// TIA Portal V17 export
// export: Created 2025-03-07T09:18:18.4685776Z, ExportSetting WithDefaults, DisplayName Totally Integrated Automation Portal, DisplayVersion V17 Update 8, DisplayName TIA Portal Openness, DisplayVersion V17 Update 8, DisplayName TIA Portal Version Control Interface, DisplayVersion V17, DisplayName SINAMICS Startdrive Advanced, DisplayVersion V17 SP2, DisplayName SINAMICS Startdrive G110M, G120, G120C, G120D, G120P, G115D, DisplayVersion V17 SP2, DisplayName SINAMICS Startdrive G130, G150, S120, S150, SINAMICS MV, S210, DisplayVersion V17 SP2, DisplayName STEP 7 Professional, DisplayVersion V17 Update 8, DisplayName SINUMERIK ONE STEP 7 Toolbox, DisplayVersion V17 Update 12, DisplayName SINUMERIK 840D sl STEP 7 Toolbox, DisplayVersion V17 Update 12, DisplayName STEP 7 Safety, DisplayVersion V17 Update 6, DisplayName WinCC Advanced, DisplayVersion V17 Update 8
FUNCTION_BLOCK "FB1401_PNEUMATIC_SYSTEM"   // FB1401, LAD
{ S7_Optimized_Access := 'FALSE' }
AUTHOR : ETXETAR
VERSION : 1.0
// stored: AutoNumber false, IsIECCheckEnabled false, SetENOAutomatically false, UDAEnableTagReadback false
   VAR_INPUT
      OPTIONS_0 : Byte := 2#0000_0000;   // OPTIONS 0
      OPTIONS_1 : Byte := 2#0000_0000;   // OPTIONS 1
      OPTIONS_2 : Byte := 2#0000_0000;   // OPTIONS 1
      PRESSURE : Bool;   // PRESSURE INPUT
      DRIVE_UNBLOCKED : Bool;   // DRIVE UNBLOCKED INPUT
      CONNECTION_1_SENSOR : Bool;   // CONNECTION 1 SENSOR INPUT
      CONNECTION_2_SENSOR : Bool;   // CONNECTION 2 SENSOR INPUT
      FLOW_SENSOR : UInt;
      TEMPERATURE_SENSOR : UInt;
      PRESSURIZED : Bool;   // PRESSURIZED INPUT
      U01_GRIPPER_PRESSURIZED : Bool;   // UNIT 01 GRIPPER PRESSURIZED INPUT
      U01_LABERINT_PRESSURIZED : Bool;   // UNIT 01 LABERINT PRESSURIZED INPUT
      U01_UPPER_TABLE_PRESSURIZED : Bool;   // UNIT 01 UPPER TABLE PRESSURIZED INPUT
      U01_LOWER_TABLE_PRESSURIZED : Bool;   // UNIT 01 LOWER TABLE PRESSURIZED INPUT
      U01_CART_X_PRESSURIZED : Bool;   // UNIT 01 AXIS X CART PRESSURIZED INPUT
      U01_STA_3_MEAS_PRESSURIZED : Bool;   // UNIT 01 STATION 3 MEASURMENT UNIT PRESSURIZED INPUT
      U02_GRIPPER_PRESSURIZED : Bool;   // UNIT 02 GRIPPER PRESSURIZED INPUT
      U02_LABERINT_PRESSURIZED : Bool;   // UNIT 02 LABERINT PRESSURIZED INPUT
      U02_UPPER_TABLE_PRESSURIZED : Bool;   // UNIT 02 UPPER TABLE PRESSURIZED INPUT
      U02_LOWER_TABLE_PRESSURIZED : Bool;   // UNIT 02 LOWER TABLEPRESSURIZED INPUT
      U02_CART_X_PRESSURIZED : Bool;   // UNIT 02 AXIS X CART PRESSURIZED INPUT
      U02_STA_3_MEAS_PRESSURIZED : Bool;   // UNIT 02 STATION 3 MEASURMENT UNIT PRESSURIZED INPUT
      HMI_REQ_LINE : Bool;   // HMI REQUEST LINE
   END_VAR
   VAR_OUTPUT
      HMI_POWER_UP_COND_OFF : Bool;   // HMI POWER UP CONDITIONS OFF
      HMI_POWER_UP_COND_ON : Bool;   // HMI POWER UP CONDITIONS ON
      HMI_POWER_UP_EXECU_LEFT : Bool;   // HMI POWER UP EXECUTABLE LEFT
      HMI_POWER_UP_EXECU_RIGHT : Bool;   // HMI POWER UP EXECUTABLE RIGHT
      MAIN_VALVE : Bool;   // MAIN VALVE OUTPUT
      CONNECTION_1 : Bool;   // CONNECTION 1 OUTPUT
      CONNECTION_2 : Bool;   // CONNECTION 2 OUTPUT
      PRESSURIZATION_ON : Bool;   // PRESSURIZATION ON OUTPUT
      PRESSURIZATION_OFF : Bool;   // PRESSURIZATION OFF OUTPUT
      DRIVE_UNBLOCK : Bool;   // DRIVE UNBLOCK OUTPUT
   END_VAR
   VAR DB_SPECIFIC
      AIR_FLOW_VALUE : Real;   // AIR FLOW INPUT
      TEMPERATURE_VALUE : Real;   // TEMPERATURE INPUT VALUE
      PRESS_NOT_REACHED_ALARM : Bool;   // PRESSURE NOT REACHED ALARM
      PRESS_SWITCH_ALARM : Bool;   // PRESSURE SWITCH ALARM
      PRESS_MISSING_ALARM : Bool;   // PRESSURE MISSING ALARM
      CONNECTION_SENSOR_1_ALARM : Bool;   // CONNECTION SENSOR 1 ALARM
      CONNECTION_SENSOR_2_ALARM : Bool;   // CONNECTION SENSOR 2 ALARM
      UNBLOCK_DRIVE_PRESS_ALARM : Bool;   // UNBLOCK DRIVE PRESSURE ALARM
      UNBLOCK_DRIVE_PRESS_SWITCH_ALARM : Bool;   // UNBLOCK DRIVE PRESSURE SWITCH ALARM
      PRESSURIZATION_ALARM : Bool;   // PRESSURIZATION ALARM
      PRESSURIZATION_SWITCH_ALARM : Bool;   // PRESSURIZATION SWITCH ALARM
      PNEUMATIC_TEMPERATURE_INPUT_ALARM : Bool;   // PNEUMATIC INPUT TEMPERATURE ALARM
      PNEUMATIC_FLOW_INPUT_ALARM : Bool;   // PNEUMATIC INPUT FLOW ALARM
      U01_GRIPPER_PRESSURIZATION_ALARM : Bool;   // UNIT 01 GRIPPER PRESSURIZATION ALARM
      U01_GRIPPER_PRESSURIZATION_SWITCH_ALARM : Bool;   // UNIT 01 GRIPPER PRESSURIZATION SWITCH ALARM
      U01_LABERINT_PRESSURIZATION_ALARM : Bool;   // UNIT 01 LABERINT PRESSURIZATION ALARM
      U01_LABERINT_PRESSURIZATION_SWITCH_ALARM : Bool;   // UNIT 01 LABERINT PRESSURIZATION SWITCH ALARM
      U01_UPPER_TABLE_PRESSURIZATION_ALARM : Bool;   // UNIT 01 UPPER TABLE PRESSURIZATION ALARM
      U01_UPPER_TABLE_PRESSURIZATION_SWITCH_ALARM : Bool;   // UNIT 01 UPPER TABLE PRESSURIZATION SWITCH ALARM
      U01_LOWER_TABLE_PRESSURIZATION_ALARM : Bool;   // UNIT 01 LOWER TABLE PRESSURIZATION ALARM
      U01_LOWER_TABLE_PRESSURIZATION_SWITCH_ALARM : Bool;   // UNIT 01 LOWER TABLE PRESSURIZATION SWITCH ALARM
      U01_CART_AXIS_X_PRESSURIZATION_ALARM : Bool;   // UNIT 01 CART AXIS X PRESSURIZATION ALARM
      U01_CART_AXIS_X_PRESSURIZATION_SWITCH_ALARM : Bool;   // UNIT 01 CART AXIS X PRESSURIZATION SWITCH ALARM
      U01_STA_3_MEAS_PRESSURIZATION_ALARM : Bool;   // UNIT 01 STATION 3 MEASUREMENT UNIT PRESSURIZATION ALARM
      U01_STA_3_MEAS_PRESSURIZATION_SWITCH_ALARM : Bool;   // UNIT 01 STATION 3 MEASUREMENT UNIT PRESSURIZATION SWITCH ALARM
      U02_GRIPPER_PRESSURIZATION_ALARM : Bool;   // UNIT 02 GRIPPER PRESSURIZATION ALARM
      U02_GRIPPER_PRESSURIZATION_SWITCH_ALARM : Bool;   // UNIT 02 GRIPPER PRESSURIZATION SWITCH ALARM
      U02_LABERINT_PRESSURIZATION_ALARM : Bool;   // UNIT 02 LABERINT PRESSURIZATION ALARM
      U02_LABERINT_PRESSURIZATION_SWITCH_ALARM : Bool;   // UNIT 02 LABERINT PRESSURIZATION SWITCH ALARM
      U02_UPPER_TABLE_PRESSURIZATION_ALARM : Bool;   // UNIT 02 UPPER TABLE PRESSURIZATION ALARM
      U02_UPPER_TABLE_PRESSURIZATION_SWITCH_ALARM : Bool;   // UNIT 02 UPPER TABLE PRESSURIZATION SWITCH ALARM
      U02_LOWER_TABLE_PRESSURIZATION_ALARM : Bool;   // UNIT 02 LOWER TABLE PRESSURIZATION ALARM
      U02_LOWER_TABLE_PRESSURIZATION_SWITCH_ALARM : Bool;   // UNIT 02 LOWER TABLE PRESSURIZATION SWITCH ALARM
      U02_CART_AXIS_X_PRESSURIZATION_ALARM : Bool;   // UNIT 02 CART AXIS X PRESSURIZATION ALARM
      U02_CART_AXIS_X_PRESSURIZATION_SWITCH_ALARM : Bool;   // UNIT 02 CART AXIS X PRESSURIZATION SWITCH ALARM
      U02_STA_3_MEAS_PRESSURIZATION_ALARM : Bool;   // UNIT 02 STATION 3 MEASUREMENT UNIT PRESSURIZATION ALARM
      U02_STA_3_MEAS_PRESSURIZATION_SWITCH_ALARM : Bool;   // UNIT 02 STATION 3 MEASUREMENT UNIT PRESSURIZATION SWITCH ALARM
      SWITCH_ON_GENERAL_CONDITIONS : Bool;   // SWITCH ON GENERAL CONDITIONS
      SWITCH_ON_INITIAL_CONDITIONS : Bool;   // SWITCH ON INITIAL CONDITIONS
      SWITCH_ON_MANUAL_REQUEST : Bool;   // SWITCH ON MANUAL REQUEST
      SWITCH_ON_AUTO_REQUEST : Bool;   // SWITCH ON AUTO REQUEST
      SWITCH_ON_GLOBAL_REQUEST : Bool;   // SWITCH ON GLOBAL REQUEST
      SWITCH_ON_COMMAND : Bool;   // SWITCH ON COMMAND
      SWITCH_ON : Bool;   // SWITCH ON
      IN_SERVICE : Bool;   // IN SERVICE
      SWITCH_OFF_GENERAL_CONDITIONS : Bool;   // SWITCH OFF GENERAL CONDITIONS
      SWITCH_OFF_INITIAL_CONDITIONS : Bool;   // SWITCH OFF INITIAL CONDITIONS
      SWITCH_OFF_MANUAL_REQUEST : Bool;   // SWITCH OFF MANUAL REQUEST
      SWITCH_OFF_AUTO_REQUEST : Bool;   // SWITCH OFF AUTO REQUEST
      SWITCH_OFF_GLOBAL_REQUEST : Bool;   // SWITCH OFF GLOBAL REQUEST
      SWITCH_OFF_COMMAND : Bool;   // SWITCH OFF COMMAND
      SWITCH_OFF : Bool;   // SWITCH OFF
      OUT_OF_SERVICE : Bool;   // OUT OF SERVICE
      MANUAL_REQUEST_HELP : Bool;   // MANUAL REQUEST HELP
      SWITCH_ON_GENERAL_CONDITION_HELP : Bool;   // SWITCH ON GENERAL CONDITION HELP
      SWITCH_ON_INITIAL_CONDITION_HELP : Bool;   // SWITCH ON INITIAL CONDITION HELP
      SWITCH_OFF_GENERAL_CONDITION_HELP : Bool;   // SWITCH OFF GENERAL CONDITION HELP
      SWITCH_OFF_INITIAL_CONDITION_HELP : Bool;   // SWITCH OFF INITIAL CONDITION HELP
      ANY_ACTIVE_ALARM : Bool;   // ANY ACTIVE ALARM
      IS_ALARMS : Bool;   // IMMEDIATE STOP ALARMS
      SEOC_ALARMS : Bool;   // STOP END OF CYCLE ALARMS
      WARNINGS : Bool;   // WARNINGS
      WARNINGS_GONE : Bool;   // WARNINGS GONE
      TIMER_PRESSURE_ALARM : TON_TIME;   // PRESSURE TIMER
      TIMER_PRESSURE_SWITCH_ALARM : TON_TIME;   // PRESSURE SWITCH TIMER
      TIMER_PRESSURE_MISSING_ALARM : TON_TIME;   // PRESSURE MISSING TIMER
      TIMER_CONNECTION_SENSOR_1_ALARM : TON_TIME;   // CONNECTION SENSOR 1 TIMER
      TIMER_CONNECTION_SENSOR_1_SWITCH_ALARM : TON_TIME;   // CONNECTION SENSOR 1 SWITCH TIMER
      TIMER_CONNECTION_SENSOR_2_ALARM : TON_TIME;   // CONNECTION SENSOR 2 TIMER
      TIMER_CONNECTION_SENSOR_2_SWITCH_ALARM : TON_TIME;   // CONNECTION SENSOR 2 SWITCH TIMER
      TIMER_DRIVE_PRESSURE_UNBLOCK_ALARM : TON_TIME;   // DRIVE PRESSURE UNBLOCK TIMER
      TIMER_DRIVE_PRESSURE_UNBLOCK_SWITCH_ALARM : TON_TIME;   // DRIVE PRESSURE UNBLOCK SWITCH TIMER
      TIMER_PRESSURE_ON_DEVICES : TON_TIME;   // PRESSURE ON DEVICES TIMER
      TIMER_PRESSURE_OFF_DEVICES : TON_TIME;   // PRESSURE OFF DEVICES TIMER
      TIMER_PRESSURIZATION_OFF_DELAY { S7_SetPoint := 'True'} : TOF_TIME;
   END_VAR
   VAR_TEMP
      INPUTS_MASK : Byte;   // INPUT MASK
      O_BYTE_0 : Struct   // OPTIONS BYTE 0
         PRESSURE_PRESENT : Bool;   // PRESSURE PRESENT OPTION
         CONNECTION_SENSOR_1 : Bool;   // CONNECTION SENSOR 1 OPTION
         CONNECTION_SENSOR_2 : Bool;   // CONNECTION SENSOR 2 OPTION
         UNBLOCK_DRIVE_VALVE : Bool;   // DRIVE VALVE OPTION
         PRESSURIZED : Bool;   // PRESSURIZED OPTION
         U01_GRIPPER_PRESSURIZED : Bool;   // UNIT 01 GRIPPER PRESSURIZED OPTION
         U01_LABERINT_PRESSURIZED : Bool;   // UNIT 01 LABERINT PRESSURIZED OPTION
         U01_UPPER_TABLE_PRESSURIZED : Bool;   // UNIT 01 UPPER TABLE PRESSURIZED OPTION
      END_STRUCT;
      O_BYTE_1 : Struct   // OPTIONS BYTE 1
         U01_LOWER_TABLE_PRESSURIZED : Bool;   // UNIT 01 LOWER TABLE PRESSURIZED OPTION
         U01_X_CART_PRESSURIZED : Bool;   // UNIT 01 AXIS X CART PRESSURIZED OPTION
         U01_STA_3_MEAS_PRESSURIZED : Bool;   // UNIT 01 STATION 3 MEASUREMENT PRESSURIZED OPTION
         U01_STA_4_MEAS_PRESSURIZED : Bool;   // UNIT 01 STATION 4 MEASUREMENT PRESSURIZED OPTION
         U02_GRIPPER_PRESSURIZED : Bool;   // UNIT 02 GRIPPER PRESSURIZED OPTION
         U02_LABERINT_PRESSURIZED : Bool;   // UNIT 02 LABERINT PRESSURIZED OPTION
         U02_UPPER_TABLE_PRESSURIZED : Bool;   // UNIT 02 UPPER TABLE PRESSURIZED OPTION
         U02_LOWER_TABLE_PRESSURIZED : Bool;   // UNIT 02 LOWER TABLE PRESSURIZED OPTION
      END_STRUCT;
      O_BYTE_2 : Struct   // OPTIONS BYTE 1
         U02_X_CART_PRESSURIZED : Bool;   // UNIT 02 AXIS X CART PRESSURIZED OPTION
         U02_STA_3_MEAS_PRESSURIZED : Bool;   // UNIT 02 STATION 3 MEASUREMENT PRESSURIZED OPTION
         U02_STA_4_MEAS_PRESSURIZED : Bool;   // UNIT 02 STATION 4 MEASUREMENT PRESSURIZED OPTION
         INPUT_FLOW_OPTION : Bool;   // INPUT FLOW OPTION
         INPUT_TEMPERATURE_OPTION : Bool;   // INPUT TEMPERATURE OPTION
         SPARE_5 : Bool;   // SPARE OPTION
         SPARE_6 : Bool;   // SPARE OPTION
         SPARE_7 : Bool;   // SPARE OPTION
      END_STRUCT;
      TEMPERATURE_TEMP : UInt;   // TEMPERATURE TEMPORAL
      PRESSURE_ON_DELAYED : Bool;   // PRESSURE ON DELAYED
      PRESSURE_OFF_DELAYED : Bool;   // PRESSURE OFF DELAYED
      DB_NUMBER : DInt;   // DB NUMBER FOR ALARM DECODING
   END_VAR
   // TIMER_PRESSURE_ALARM.PT := T#1M;
   // TIMER_PRESSURE_SWITCH_ALARM.PT := T#1M;
   // TIMER_PRESSURE_MISSING_ALARM.PT := T#1s;
   // TIMER_CONNECTION_SENSOR_1_ALARM.PT := T#1s;
   // TIMER_CONNECTION_SENSOR_1_SWITCH_ALARM.PT := T#1s;
   // TIMER_CONNECTION_SENSOR_2_ALARM.PT := T#1s;
   // TIMER_CONNECTION_SENSOR_2_SWITCH_ALARM.PT := T#1s;
   // TIMER_DRIVE_PRESSURE_UNBLOCK_ALARM.PT := T#3s;
   // TIMER_DRIVE_PRESSURE_UNBLOCK_SWITCH_ALARM.PT := T#3s;
   // TIMER_PRESSURE_ON_DEVICES.PT := T#5s;
   // TIMER_PRESSURE_OFF_DEVICES.PT := T#31M;
   // TIMER_PRESSURIZATION_OFF_DELAY.PT := T#30M;
   VAR_TEMP   // added for the SCL form of the ladder/FBD networks
      _w1 : Bool;
   END_VAR
BEGIN

NETWORK
TITLE = READ INSTANCE DB
      L     DINO;
      +     10#800000;
      T     #DB_NUMBER;


REGION Network 2: OPTIONS
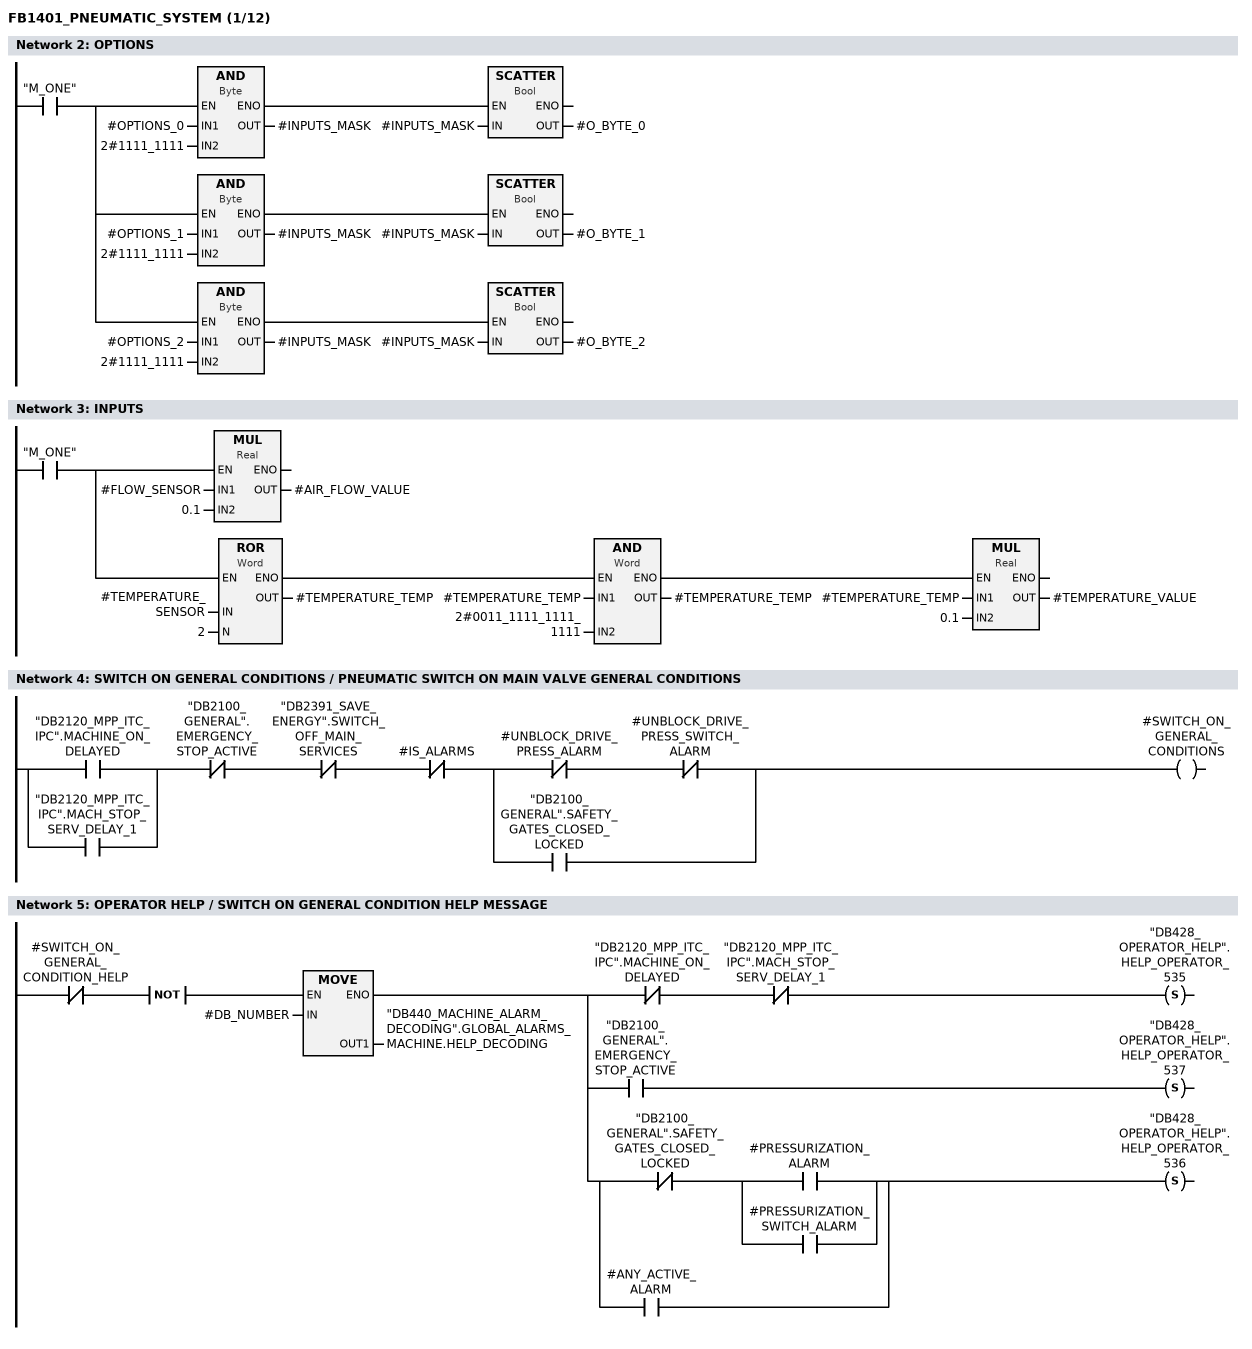
   RUNG wire#powerrail
      Contact( "M_ONE" )
      wire#w1
      { S7_Templates := "SrcType := Byte"; S7_GenerateENO := "TRUE" } And(in1 := #OPTIONS_0, in2 := 2#1111_1111, out => #INPUTS_MASK)
      { S7_Templates := "[dest_type := Bool, src_type := Byte]" } SCATTER(IN := #INPUTS_MASK, OUT => #O_BYTE_0)
   END_RUNG
   RUNG wire#w1
      { S7_Templates := "SrcType := Byte"; S7_GenerateENO := "TRUE" } And(in1 := #OPTIONS_1, in2 := 2#1111_1111, out => #INPUTS_MASK)
      { S7_Templates := "[dest_type := Bool, src_type := Byte]" } SCATTER(IN := #INPUTS_MASK, OUT => #O_BYTE_1)
   END_RUNG
   RUNG wire#w1
      { S7_Templates := "SrcType := Byte"; S7_GenerateENO := "TRUE" } And(in1 := #OPTIONS_2, in2 := 2#1111_1111, out => #INPUTS_MASK)
      { S7_Templates := "[dest_type := Bool, src_type := Byte]" } SCATTER(IN := #INPUTS_MASK, OUT => #O_BYTE_2)
   END_RUNG
   // the same network as SCL:
   IF "M_ONE" THEN #INPUTS_MASK := #OPTIONS_0 AND 2#1111_1111; END_IF;
   #_w1 := "M_ONE";
   IF #_w1 THEN
       SCATTER(IN := #INPUTS_MASK, OUT => #O_BYTE_0);
       #INPUTS_MASK := #OPTIONS_1 AND 2#1111_1111;
       SCATTER(IN := #INPUTS_MASK, OUT => #O_BYTE_1);
       #INPUTS_MASK := #OPTIONS_2 AND 2#1111_1111;
       SCATTER(IN := #INPUTS_MASK, OUT => #O_BYTE_2);
   END_IF;
END_REGION

REGION Network 3: INPUTS
   IF "M_ONE" THEN
       #AIR_FLOW_VALUE := #FLOW_SENSOR * 0.1;
       #TEMPERATURE_TEMP := ROR(IN := #TEMPERATURE_SENSOR, N := 2);
       #TEMPERATURE_TEMP := #TEMPERATURE_TEMP AND 2#0011_1111_1111_1111;
       #TEMPERATURE_VALUE := #TEMPERATURE_TEMP * 0.1;
   END_IF;
END_REGION

REGION Network 4: SWITCH ON GENERAL CONDITIONS / PNEUMATIC SWITCH ON MAIN VALVE GENERAL CONDITIONS
   RUNG wire#powerrail
      Contact( "DB2120_MPP_ITC_IPC".MACHINE_ON_DELAYED )
      wire#w1
      I_Contact( "DB2100_GENERAL".EMERGENCY_STOP_ACTIVE )
      I_Contact( "DB2391_SAVE_ENERGY".SWITCH_OFF_MAIN_SERVICES )
      I_Contact( #IS_ALARMS )
      wire#w2
      I_Contact( #UNBLOCK_DRIVE_PRESS_ALARM )
      I_Contact( #UNBLOCK_DRIVE_PRESS_SWITCH_ALARM )
      wire#w3
      Coil( #SWITCH_ON_GENERAL_CONDITIONS )
   END_RUNG
   RUNG wire#powerrail
      Contact( "DB2120_MPP_ITC_IPC".MACH_STOP_SERV_DELAY_1 )
   END_RUNG wire#w1
   RUNG wire#w2
      Contact( "DB2100_GENERAL".SAFETY_GATES_CLOSED_LOCKED )
   END_RUNG wire#w3
   // the same network as SCL:
   #SWITCH_ON_GENERAL_CONDITIONS := ("DB2120_MPP_ITC_IPC".MACHINE_ON_DELAYED OR "DB2120_MPP_ITC_IPC".MACH_STOP_SERV_DELAY_1) AND NOT "DB2100_GENERAL".EMERGENCY_STOP_ACTIVE AND NOT "DB2391_SAVE_ENERGY".SWITCH_OFF_MAIN_SERVICES AND NOT #IS_ALARMS AND ((NOT #UNBLOCK_DRIVE_PRESS_ALARM AND NOT #UNBLOCK_DRIVE_PRESS_SWITCH_ALARM) OR "DB2100_GENERAL".SAFETY_GATES_CLOSED_LOCKED);
END_REGION

REGION Network 5: OPERATOR HELP / SWITCH ON GENERAL CONDITION HELP MESSAGE
   RUNG wire#powerrail
      I_Contact( #SWITCH_ON_GENERAL_CONDITION_HELP )
      Not()
      { S7_GenerateENO := "TRUE" } Move(in := #DB_NUMBER, out1 => "DB440_MACHINE_ALARM_DECODING".GLOBAL_ALARMS_MACHINE.HELP_DECODING)
      wire#w1
      I_Contact( "DB2120_MPP_ITC_IPC".MACHINE_ON_DELAYED )
      I_Contact( "DB2120_MPP_ITC_IPC".MACH_STOP_SERV_DELAY_1 )
      S_Coil( "DB428_OPERATOR_HELP".HELP_OPERATOR_535 )
   END_RUNG
   RUNG wire#w1
      Contact( "DB2100_GENERAL".EMERGENCY_STOP_ACTIVE )
      S_Coil( "DB428_OPERATOR_HELP".HELP_OPERATOR_537 )
   END_RUNG
   RUNG wire#w1
      I_Contact( "DB2100_GENERAL".SAFETY_GATES_CLOSED_LOCKED )
      wire#w2
      Contact( #PRESSURIZATION_ALARM )
      wire#w3
      S_Coil( "DB428_OPERATOR_HELP".HELP_OPERATOR_536 )
   END_RUNG
   RUNG wire#w2
      Contact( #PRESSURIZATION_SWITCH_ALARM )
   END_RUNG wire#w3
   RUNG wire#w1
      Contact( #ANY_ACTIVE_ALARM )
   END_RUNG wire#w3
   // the same network as SCL:
   // ENO of a box is taken as its EN; it also drops when the box reports an error
   #_w1 := NOT (NOT #SWITCH_ON_GENERAL_CONDITION_HELP);
   IF #_w1 THEN "DB440_MACHINE_ALARM_DECODING".GLOBAL_ALARMS_MACHINE.HELP_DECODING := #DB_NUMBER; END_IF;
   IF #_w1 AND NOT "DB2120_MPP_ITC_IPC".MACHINE_ON_DELAYED AND NOT "DB2120_MPP_ITC_IPC".MACH_STOP_SERV_DELAY_1 THEN
       "DB428_OPERATOR_HELP".HELP_OPERATOR_535 := TRUE;
   END_IF;
   IF #_w1 AND "DB2100_GENERAL".EMERGENCY_STOP_ACTIVE THEN
       "DB428_OPERATOR_HELP".HELP_OPERATOR_537 := TRUE;
   END_IF;
   IF #_w1 AND ((NOT "DB2100_GENERAL".SAFETY_GATES_CLOSED_LOCKED AND (#PRESSURIZATION_ALARM OR #PRESSURIZATION_SWITCH_ALARM)) OR #ANY_ACTIVE_ALARM) THEN
       "DB428_OPERATOR_HELP".HELP_OPERATOR_536 := TRUE;
   END_IF;
END_REGION

REGION Network 6: SWITCH ON INITIAL CONDITIONS
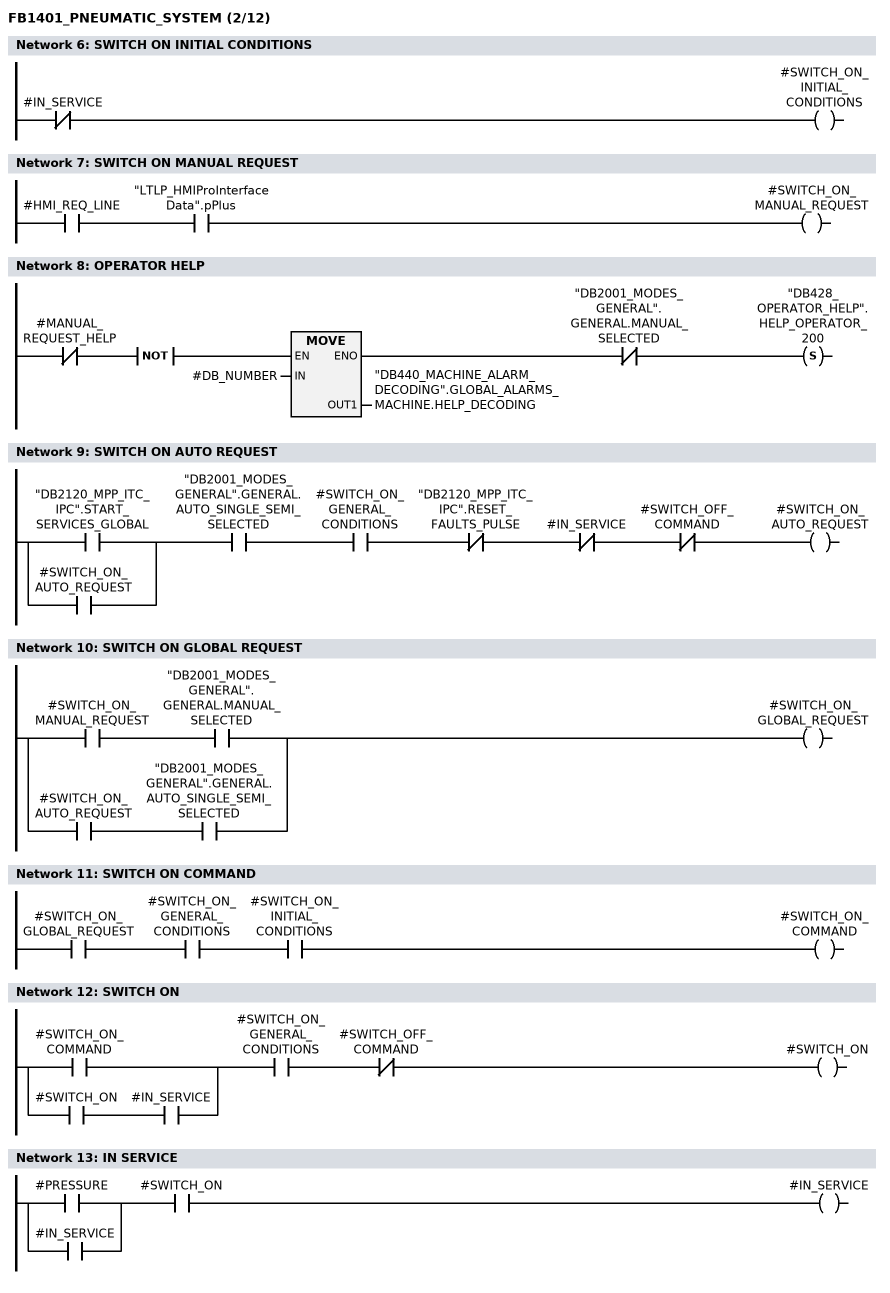
   RUNG wire#powerrail
      I_Contact( #IN_SERVICE )
      Coil( #SWITCH_ON_INITIAL_CONDITIONS )
   END_RUNG
   // the same network as SCL:
   #SWITCH_ON_INITIAL_CONDITIONS := NOT #IN_SERVICE;
END_REGION

REGION Network 7: SWITCH ON MANUAL REQUEST
   RUNG wire#powerrail
      Contact( #HMI_REQ_LINE )
      Contact( "LTLP_HMIProInterfaceData".pPlus )
      Coil( #SWITCH_ON_MANUAL_REQUEST )
   END_RUNG
   // the same network as SCL:
   #SWITCH_ON_MANUAL_REQUEST := #HMI_REQ_LINE AND "LTLP_HMIProInterfaceData".pPlus;
END_REGION

REGION Network 8: OPERATOR HELP
   RUNG wire#powerrail
      I_Contact( #MANUAL_REQUEST_HELP )
      Not()
      { S7_GenerateENO := "TRUE" } Move(in := #DB_NUMBER, out1 => "DB440_MACHINE_ALARM_DECODING".GLOBAL_ALARMS_MACHINE.HELP_DECODING)
      I_Contact( "DB2001_MODES_GENERAL".GENERAL.MANUAL_SELECTED )
      S_Coil( "DB428_OPERATOR_HELP".HELP_OPERATOR_200 )
   END_RUNG
   // the same network as SCL:
   // ENO of a box is taken as its EN; it also drops when the box reports an error
   #_w1 := NOT (NOT #MANUAL_REQUEST_HELP);
   IF #_w1 THEN "DB440_MACHINE_ALARM_DECODING".GLOBAL_ALARMS_MACHINE.HELP_DECODING := #DB_NUMBER; END_IF;
   IF #_w1 AND NOT "DB2001_MODES_GENERAL".GENERAL.MANUAL_SELECTED THEN
       "DB428_OPERATOR_HELP".HELP_OPERATOR_200 := TRUE;
   END_IF;
END_REGION

REGION Network 9: SWITCH ON AUTO REQUEST
   RUNG wire#powerrail
      Contact( "DB2120_MPP_ITC_IPC".START_SERVICES_GLOBAL )
      wire#w1
      Contact( "DB2001_MODES_GENERAL".GENERAL.AUTO_SINGLE_SEMI_SELECTED )
      Contact( #SWITCH_ON_GENERAL_CONDITIONS )
      I_Contact( "DB2120_MPP_ITC_IPC".RESET_FAULTS_PULSE )
      I_Contact( #IN_SERVICE )
      I_Contact( #SWITCH_OFF_COMMAND )
      Coil( #SWITCH_ON_AUTO_REQUEST )
   END_RUNG
   RUNG wire#powerrail
      Contact( #SWITCH_ON_AUTO_REQUEST )
   END_RUNG wire#w1
   // the same network as SCL:
   #SWITCH_ON_AUTO_REQUEST := ("DB2120_MPP_ITC_IPC".START_SERVICES_GLOBAL OR #SWITCH_ON_AUTO_REQUEST) AND "DB2001_MODES_GENERAL".GENERAL.AUTO_SINGLE_SEMI_SELECTED AND #SWITCH_ON_GENERAL_CONDITIONS AND NOT "DB2120_MPP_ITC_IPC".RESET_FAULTS_PULSE AND NOT #IN_SERVICE AND NOT #SWITCH_OFF_COMMAND;
END_REGION

REGION Network 10: SWITCH ON GLOBAL REQUEST
   RUNG wire#powerrail
      Contact( #SWITCH_ON_MANUAL_REQUEST )
      Contact( "DB2001_MODES_GENERAL".GENERAL.MANUAL_SELECTED )
      wire#w1
      Coil( #SWITCH_ON_GLOBAL_REQUEST )
   END_RUNG
   RUNG wire#powerrail
      Contact( #SWITCH_ON_AUTO_REQUEST )
      Contact( "DB2001_MODES_GENERAL".GENERAL.AUTO_SINGLE_SEMI_SELECTED )
   END_RUNG wire#w1
   // the same network as SCL:
   #SWITCH_ON_GLOBAL_REQUEST := (#SWITCH_ON_MANUAL_REQUEST AND "DB2001_MODES_GENERAL".GENERAL.MANUAL_SELECTED) OR (#SWITCH_ON_AUTO_REQUEST AND "DB2001_MODES_GENERAL".GENERAL.AUTO_SINGLE_SEMI_SELECTED);
END_REGION

REGION Network 11: SWITCH ON COMMAND
   RUNG wire#powerrail
      Contact( #SWITCH_ON_GLOBAL_REQUEST )
      Contact( #SWITCH_ON_GENERAL_CONDITIONS )
      Contact( #SWITCH_ON_INITIAL_CONDITIONS )
      Coil( #SWITCH_ON_COMMAND )
   END_RUNG
   // the same network as SCL:
   #SWITCH_ON_COMMAND := #SWITCH_ON_GLOBAL_REQUEST AND #SWITCH_ON_GENERAL_CONDITIONS AND #SWITCH_ON_INITIAL_CONDITIONS;
END_REGION

REGION Network 12: SWITCH ON
   RUNG wire#powerrail
      Contact( #SWITCH_ON_COMMAND )
      wire#w1
      Contact( #SWITCH_ON_GENERAL_CONDITIONS )
      I_Contact( #SWITCH_OFF_COMMAND )
      Coil( #SWITCH_ON )
   END_RUNG
   RUNG wire#powerrail
      Contact( #SWITCH_ON )
      Contact( #IN_SERVICE )
   END_RUNG wire#w1
   // the same network as SCL:
   #SWITCH_ON := (#SWITCH_ON_COMMAND OR (#SWITCH_ON AND #IN_SERVICE)) AND #SWITCH_ON_GENERAL_CONDITIONS AND NOT #SWITCH_OFF_COMMAND;
END_REGION

REGION Network 13: IN SERVICE
   RUNG wire#powerrail
      Contact( #PRESSURE )
      wire#w1
      Contact( #SWITCH_ON )
      Coil( #IN_SERVICE )
   END_RUNG
   RUNG wire#powerrail
      Contact( #IN_SERVICE )
   END_RUNG wire#w1
   // the same network as SCL:
   #IN_SERVICE := (#PRESSURE OR #IN_SERVICE) AND #SWITCH_ON;
END_REGION

REGION Network 14: SWITCH OFF GENERAL CONDITIONS
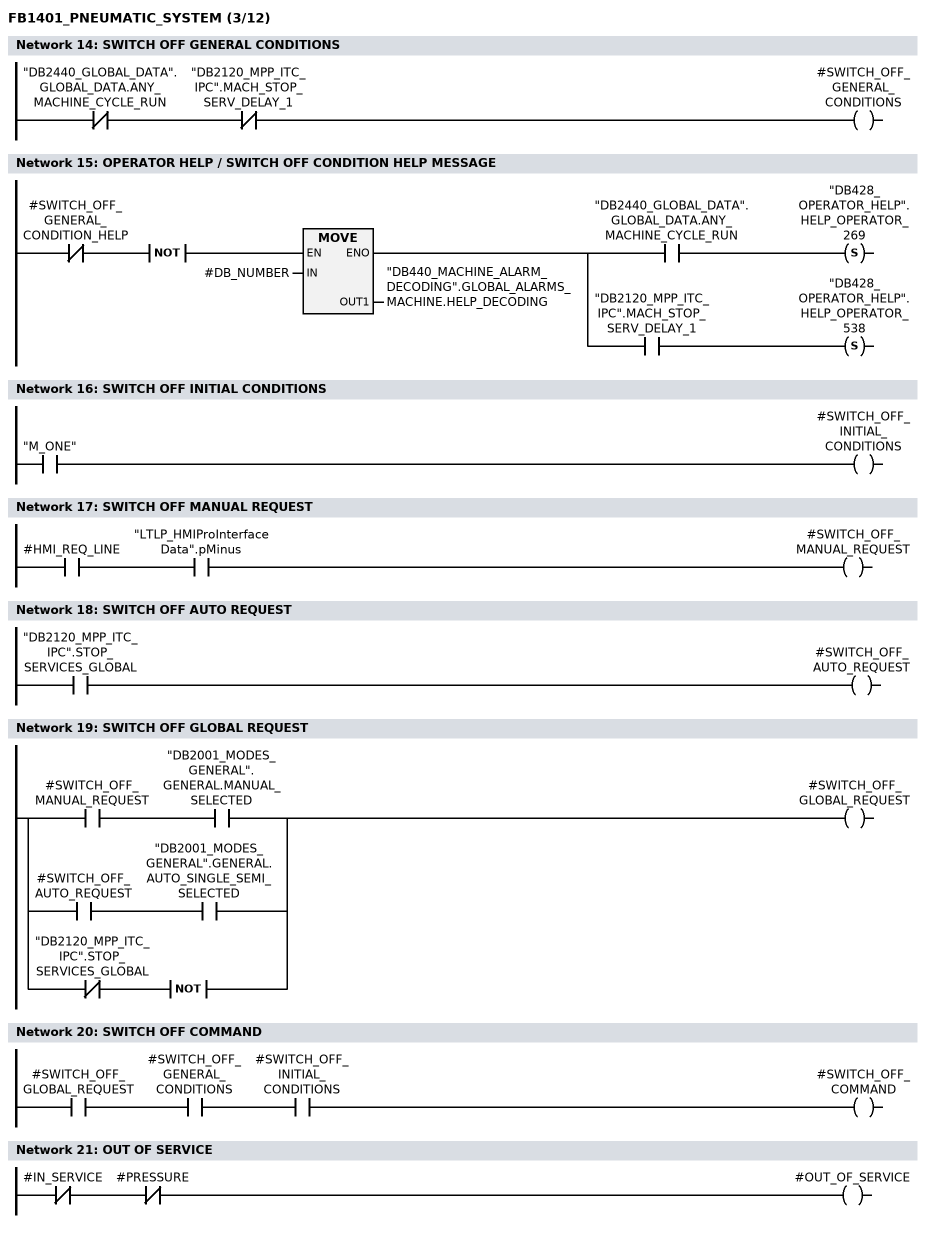
   RUNG wire#powerrail
      I_Contact( "DB2440_GLOBAL_DATA".GLOBAL_DATA.ANY_MACHINE_CYCLE_RUN )
      I_Contact( "DB2120_MPP_ITC_IPC".MACH_STOP_SERV_DELAY_1 )
      Coil( #SWITCH_OFF_GENERAL_CONDITIONS )
   END_RUNG
   // the same network as SCL:
   #SWITCH_OFF_GENERAL_CONDITIONS := NOT "DB2440_GLOBAL_DATA".GLOBAL_DATA.ANY_MACHINE_CYCLE_RUN AND NOT "DB2120_MPP_ITC_IPC".MACH_STOP_SERV_DELAY_1;
END_REGION

REGION Network 15: OPERATOR HELP / SWITCH OFF CONDITION HELP MESSAGE
   RUNG wire#powerrail
      I_Contact( #SWITCH_OFF_GENERAL_CONDITION_HELP )
      Not()
      { S7_GenerateENO := "TRUE" } Move(in := #DB_NUMBER, out1 => "DB440_MACHINE_ALARM_DECODING".GLOBAL_ALARMS_MACHINE.HELP_DECODING)
      wire#w1
      Contact( "DB2440_GLOBAL_DATA".GLOBAL_DATA.ANY_MACHINE_CYCLE_RUN )
      S_Coil( "DB428_OPERATOR_HELP".HELP_OPERATOR_269 )
   END_RUNG
   RUNG wire#w1
      Contact( "DB2120_MPP_ITC_IPC".MACH_STOP_SERV_DELAY_1 )
      S_Coil( "DB428_OPERATOR_HELP".HELP_OPERATOR_538 )
   END_RUNG
   // the same network as SCL:
   // ENO of a box is taken as its EN; it also drops when the box reports an error
   #_w1 := NOT (NOT #SWITCH_OFF_GENERAL_CONDITION_HELP);
   IF #_w1 THEN "DB440_MACHINE_ALARM_DECODING".GLOBAL_ALARMS_MACHINE.HELP_DECODING := #DB_NUMBER; END_IF;
   IF #_w1 AND "DB2440_GLOBAL_DATA".GLOBAL_DATA.ANY_MACHINE_CYCLE_RUN THEN
       "DB428_OPERATOR_HELP".HELP_OPERATOR_269 := TRUE;
   END_IF;
   IF #_w1 AND "DB2120_MPP_ITC_IPC".MACH_STOP_SERV_DELAY_1 THEN
       "DB428_OPERATOR_HELP".HELP_OPERATOR_538 := TRUE;
   END_IF;
END_REGION

REGION Network 16: SWITCH OFF INITIAL CONDITIONS
   RUNG wire#powerrail
      Contact( "M_ONE" )
      Coil( #SWITCH_OFF_INITIAL_CONDITIONS )
   END_RUNG
   // the same network as SCL:
   #SWITCH_OFF_INITIAL_CONDITIONS := "M_ONE";
END_REGION

REGION Network 17: SWITCH OFF MANUAL REQUEST
   RUNG wire#powerrail
      Contact( #HMI_REQ_LINE )
      Contact( "LTLP_HMIProInterfaceData".pMinus )
      Coil( #SWITCH_OFF_MANUAL_REQUEST )
   END_RUNG
   // the same network as SCL:
   #SWITCH_OFF_MANUAL_REQUEST := #HMI_REQ_LINE AND "LTLP_HMIProInterfaceData".pMinus;
END_REGION

REGION Network 18: SWITCH OFF AUTO REQUEST
   RUNG wire#powerrail
      Contact( "DB2120_MPP_ITC_IPC".STOP_SERVICES_GLOBAL )
      Coil( #SWITCH_OFF_AUTO_REQUEST )
   END_RUNG
   // the same network as SCL:
   #SWITCH_OFF_AUTO_REQUEST := "DB2120_MPP_ITC_IPC".STOP_SERVICES_GLOBAL;
END_REGION

REGION Network 19: SWITCH OFF GLOBAL REQUEST
   RUNG wire#powerrail
      Contact( #SWITCH_OFF_MANUAL_REQUEST )
      Contact( "DB2001_MODES_GENERAL".GENERAL.MANUAL_SELECTED )
      wire#w1
      Coil( #SWITCH_OFF_GLOBAL_REQUEST )
   END_RUNG
   RUNG wire#powerrail
      Contact( #SWITCH_OFF_AUTO_REQUEST )
      Contact( "DB2001_MODES_GENERAL".GENERAL.AUTO_SINGLE_SEMI_SELECTED )
   END_RUNG wire#w1
   RUNG wire#powerrail
      I_Contact( "DB2120_MPP_ITC_IPC".STOP_SERVICES_GLOBAL )
      Not()
   END_RUNG wire#w1
   // the same network as SCL:
   #SWITCH_OFF_GLOBAL_REQUEST := (#SWITCH_OFF_MANUAL_REQUEST AND "DB2001_MODES_GENERAL".GENERAL.MANUAL_SELECTED) OR (#SWITCH_OFF_AUTO_REQUEST AND "DB2001_MODES_GENERAL".GENERAL.AUTO_SINGLE_SEMI_SELECTED) OR NOT (NOT "DB2120_MPP_ITC_IPC".STOP_SERVICES_GLOBAL);
END_REGION

REGION Network 20: SWITCH OFF COMMAND
   RUNG wire#powerrail
      Contact( #SWITCH_OFF_GLOBAL_REQUEST )
      Contact( #SWITCH_OFF_GENERAL_CONDITIONS )
      Contact( #SWITCH_OFF_INITIAL_CONDITIONS )
      Coil( #SWITCH_OFF_COMMAND )
   END_RUNG
   // the same network as SCL:
   #SWITCH_OFF_COMMAND := #SWITCH_OFF_GLOBAL_REQUEST AND #SWITCH_OFF_GENERAL_CONDITIONS AND #SWITCH_OFF_INITIAL_CONDITIONS;
END_REGION

REGION Network 21: OUT OF SERVICE
   RUNG wire#powerrail
      I_Contact( #IN_SERVICE )
      I_Contact( #PRESSURE )
      Coil( #OUT_OF_SERVICE )
   END_RUNG
   // the same network as SCL:
   #OUT_OF_SERVICE := NOT #IN_SERVICE AND NOT #PRESSURE;
END_REGION

REGION Network 22: PRESSURE NOT REACHED ALARM / PNEUMATIC SYSTEM PRESSURE SWITCH ALARM
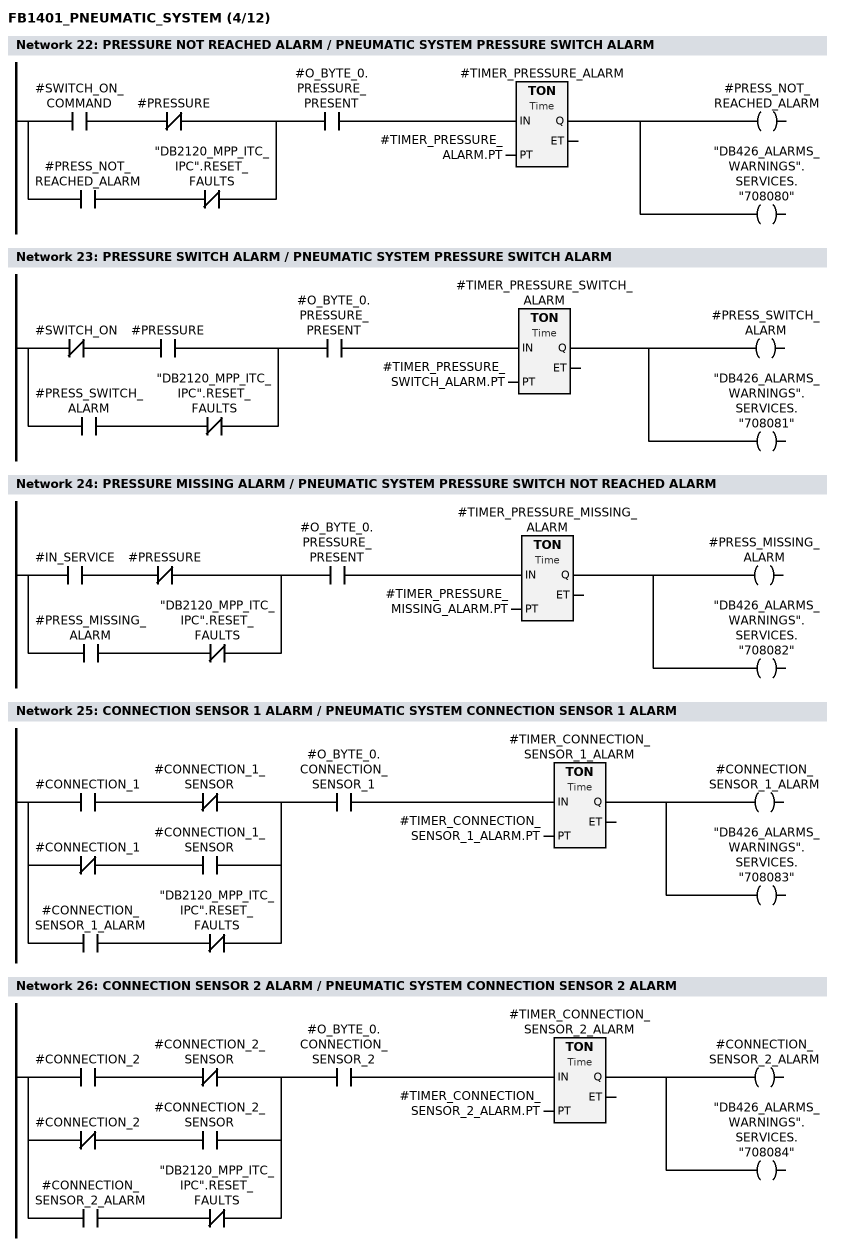
   RUNG wire#powerrail
      Contact( #SWITCH_ON_COMMAND )
      I_Contact( #PRESSURE )
      wire#w1
      Contact( #O_BYTE_0.PRESSURE_PRESENT )
      { S7_Templates := "time_type := Time" } #TIMER_PRESSURE_ALARM.TON(pt := #TIMER_PRESSURE_ALARM.PT, et =>)
      wire#w2
      Coil( #PRESS_NOT_REACHED_ALARM )
   END_RUNG
   RUNG wire#powerrail
      Contact( #PRESS_NOT_REACHED_ALARM )
      I_Contact( "DB2120_MPP_ITC_IPC".RESET_FAULTS )
   END_RUNG wire#w1
   RUNG wire#w2
      Coil( "DB426_ALARMS_WARNINGS".SERVICES."708080" )
   END_RUNG
   // the same network as SCL:
   #TIMER_PRESSURE_ALARM(IN := ((#SWITCH_ON_COMMAND AND NOT #PRESSURE) OR (#PRESS_NOT_REACHED_ALARM AND NOT "DB2120_MPP_ITC_IPC".RESET_FAULTS)) AND #O_BYTE_0.PRESSURE_PRESENT,   // TON
                         PT := #TIMER_PRESSURE_ALARM.PT);
   #PRESS_NOT_REACHED_ALARM := #TIMER_PRESSURE_ALARM.Q;
   "DB426_ALARMS_WARNINGS".SERVICES."708080" := #TIMER_PRESSURE_ALARM.Q;
END_REGION

REGION Network 23: PRESSURE SWITCH ALARM / PNEUMATIC SYSTEM PRESSURE SWITCH ALARM
   RUNG wire#powerrail
      I_Contact( #SWITCH_ON )
      Contact( #PRESSURE )
      wire#w1
      Contact( #O_BYTE_0.PRESSURE_PRESENT )
      { S7_Templates := "time_type := Time" } #TIMER_PRESSURE_SWITCH_ALARM.TON(pt := #TIMER_PRESSURE_SWITCH_ALARM.PT, et =>)
      wire#w2
      Coil( #PRESS_SWITCH_ALARM )
   END_RUNG
   RUNG wire#powerrail
      Contact( #PRESS_SWITCH_ALARM )
      I_Contact( "DB2120_MPP_ITC_IPC".RESET_FAULTS )
   END_RUNG wire#w1
   RUNG wire#w2
      Coil( "DB426_ALARMS_WARNINGS".SERVICES."708081" )
   END_RUNG
   // the same network as SCL:
   #TIMER_PRESSURE_SWITCH_ALARM(IN := ((NOT #SWITCH_ON AND #PRESSURE) OR (#PRESS_SWITCH_ALARM AND NOT "DB2120_MPP_ITC_IPC".RESET_FAULTS)) AND #O_BYTE_0.PRESSURE_PRESENT,   // TON
                           PT := #TIMER_PRESSURE_SWITCH_ALARM.PT);
   #PRESS_SWITCH_ALARM := #TIMER_PRESSURE_SWITCH_ALARM.Q;
   "DB426_ALARMS_WARNINGS".SERVICES."708081" := #TIMER_PRESSURE_SWITCH_ALARM.Q;
END_REGION

REGION Network 24: PRESSURE MISSING ALARM / PNEUMATIC SYSTEM PRESSURE SWITCH NOT REACHED ALARM
   RUNG wire#powerrail
      Contact( #IN_SERVICE )
      I_Contact( #PRESSURE )
      wire#w1
      Contact( #O_BYTE_0.PRESSURE_PRESENT )
      { S7_Templates := "time_type := Time" } #TIMER_PRESSURE_MISSING_ALARM.TON(pt := #TIMER_PRESSURE_MISSING_ALARM.PT, et =>)
      wire#w2
      Coil( #PRESS_MISSING_ALARM )
   END_RUNG
   RUNG wire#powerrail
      Contact( #PRESS_MISSING_ALARM )
      I_Contact( "DB2120_MPP_ITC_IPC".RESET_FAULTS )
   END_RUNG wire#w1
   RUNG wire#w2
      Coil( "DB426_ALARMS_WARNINGS".SERVICES."708082" )
   END_RUNG
   // the same network as SCL:
   #TIMER_PRESSURE_MISSING_ALARM(IN := ((#IN_SERVICE AND NOT #PRESSURE) OR (#PRESS_MISSING_ALARM AND NOT "DB2120_MPP_ITC_IPC".RESET_FAULTS)) AND #O_BYTE_0.PRESSURE_PRESENT,   // TON
                           PT := #TIMER_PRESSURE_MISSING_ALARM.PT);
   #PRESS_MISSING_ALARM := #TIMER_PRESSURE_MISSING_ALARM.Q;
   "DB426_ALARMS_WARNINGS".SERVICES."708082" := #TIMER_PRESSURE_MISSING_ALARM.Q;
END_REGION

REGION Network 25: CONNECTION SENSOR 1 ALARM / PNEUMATIC SYSTEM CONNECTION SENSOR 1 ALARM
   RUNG wire#powerrail
      Contact( #CONNECTION_1 )
      I_Contact( #CONNECTION_1_SENSOR )
      wire#w1
      Contact( #O_BYTE_0.CONNECTION_SENSOR_1 )
      { S7_Templates := "time_type := Time" } #TIMER_CONNECTION_SENSOR_1_ALARM.TON(pt := #TIMER_CONNECTION_SENSOR_1_ALARM.PT, et =>)
      wire#w2
      Coil( #CONNECTION_SENSOR_1_ALARM )
   END_RUNG
   RUNG wire#powerrail
      I_Contact( #CONNECTION_1 )
      Contact( #CONNECTION_1_SENSOR )
   END_RUNG wire#w1
   RUNG wire#powerrail
      Contact( #CONNECTION_SENSOR_1_ALARM )
      I_Contact( "DB2120_MPP_ITC_IPC".RESET_FAULTS )
   END_RUNG wire#w1
   RUNG wire#w2
      Coil( "DB426_ALARMS_WARNINGS".SERVICES."708083" )
   END_RUNG
   // the same network as SCL:
   #TIMER_CONNECTION_SENSOR_1_ALARM(IN := ((#CONNECTION_1 AND NOT #CONNECTION_1_SENSOR) OR (NOT #CONNECTION_1 AND #CONNECTION_1_SENSOR) OR (#CONNECTION_SENSOR_1_ALARM AND NOT "DB2120_MPP_ITC_IPC".RESET_FAULTS)) AND #O_BYTE_0.CONNECTION_SENSOR_1,   // TON
                           PT := #TIMER_CONNECTION_SENSOR_1_ALARM.PT);
   #CONNECTION_SENSOR_1_ALARM := #TIMER_CONNECTION_SENSOR_1_ALARM.Q;
   "DB426_ALARMS_WARNINGS".SERVICES."708083" := #TIMER_CONNECTION_SENSOR_1_ALARM.Q;
END_REGION

REGION Network 26: CONNECTION SENSOR 2 ALARM / PNEUMATIC SYSTEM CONNECTION SENSOR 2 ALARM
   RUNG wire#powerrail
      Contact( #CONNECTION_2 )
      I_Contact( #CONNECTION_2_SENSOR )
      wire#w1
      Contact( #O_BYTE_0.CONNECTION_SENSOR_2 )
      { S7_Templates := "time_type := Time" } #TIMER_CONNECTION_SENSOR_2_ALARM.TON(pt := #TIMER_CONNECTION_SENSOR_2_ALARM.PT, et =>)
      wire#w2
      Coil( #CONNECTION_SENSOR_2_ALARM )
   END_RUNG
   RUNG wire#powerrail
      I_Contact( #CONNECTION_2 )
      Contact( #CONNECTION_2_SENSOR )
   END_RUNG wire#w1
   RUNG wire#powerrail
      Contact( #CONNECTION_SENSOR_2_ALARM )
      I_Contact( "DB2120_MPP_ITC_IPC".RESET_FAULTS )
   END_RUNG wire#w1
   RUNG wire#w2
      Coil( "DB426_ALARMS_WARNINGS".SERVICES."708084" )
   END_RUNG
   // the same network as SCL:
   #TIMER_CONNECTION_SENSOR_2_ALARM(IN := ((#CONNECTION_2 AND NOT #CONNECTION_2_SENSOR) OR (NOT #CONNECTION_2 AND #CONNECTION_2_SENSOR) OR (#CONNECTION_SENSOR_2_ALARM AND NOT "DB2120_MPP_ITC_IPC".RESET_FAULTS)) AND #O_BYTE_0.CONNECTION_SENSOR_2,   // TON
                           PT := #TIMER_CONNECTION_SENSOR_2_ALARM.PT);
   #CONNECTION_SENSOR_2_ALARM := #TIMER_CONNECTION_SENSOR_2_ALARM.Q;
   "DB426_ALARMS_WARNINGS".SERVICES."708084" := #TIMER_CONNECTION_SENSOR_2_ALARM.Q;
END_REGION

REGION Network 27: UNBLOCK DRIVE PRESSURE ALARM / PNEUMATIC SYSTEM UNBLOCK VALVE FAULT DELAY
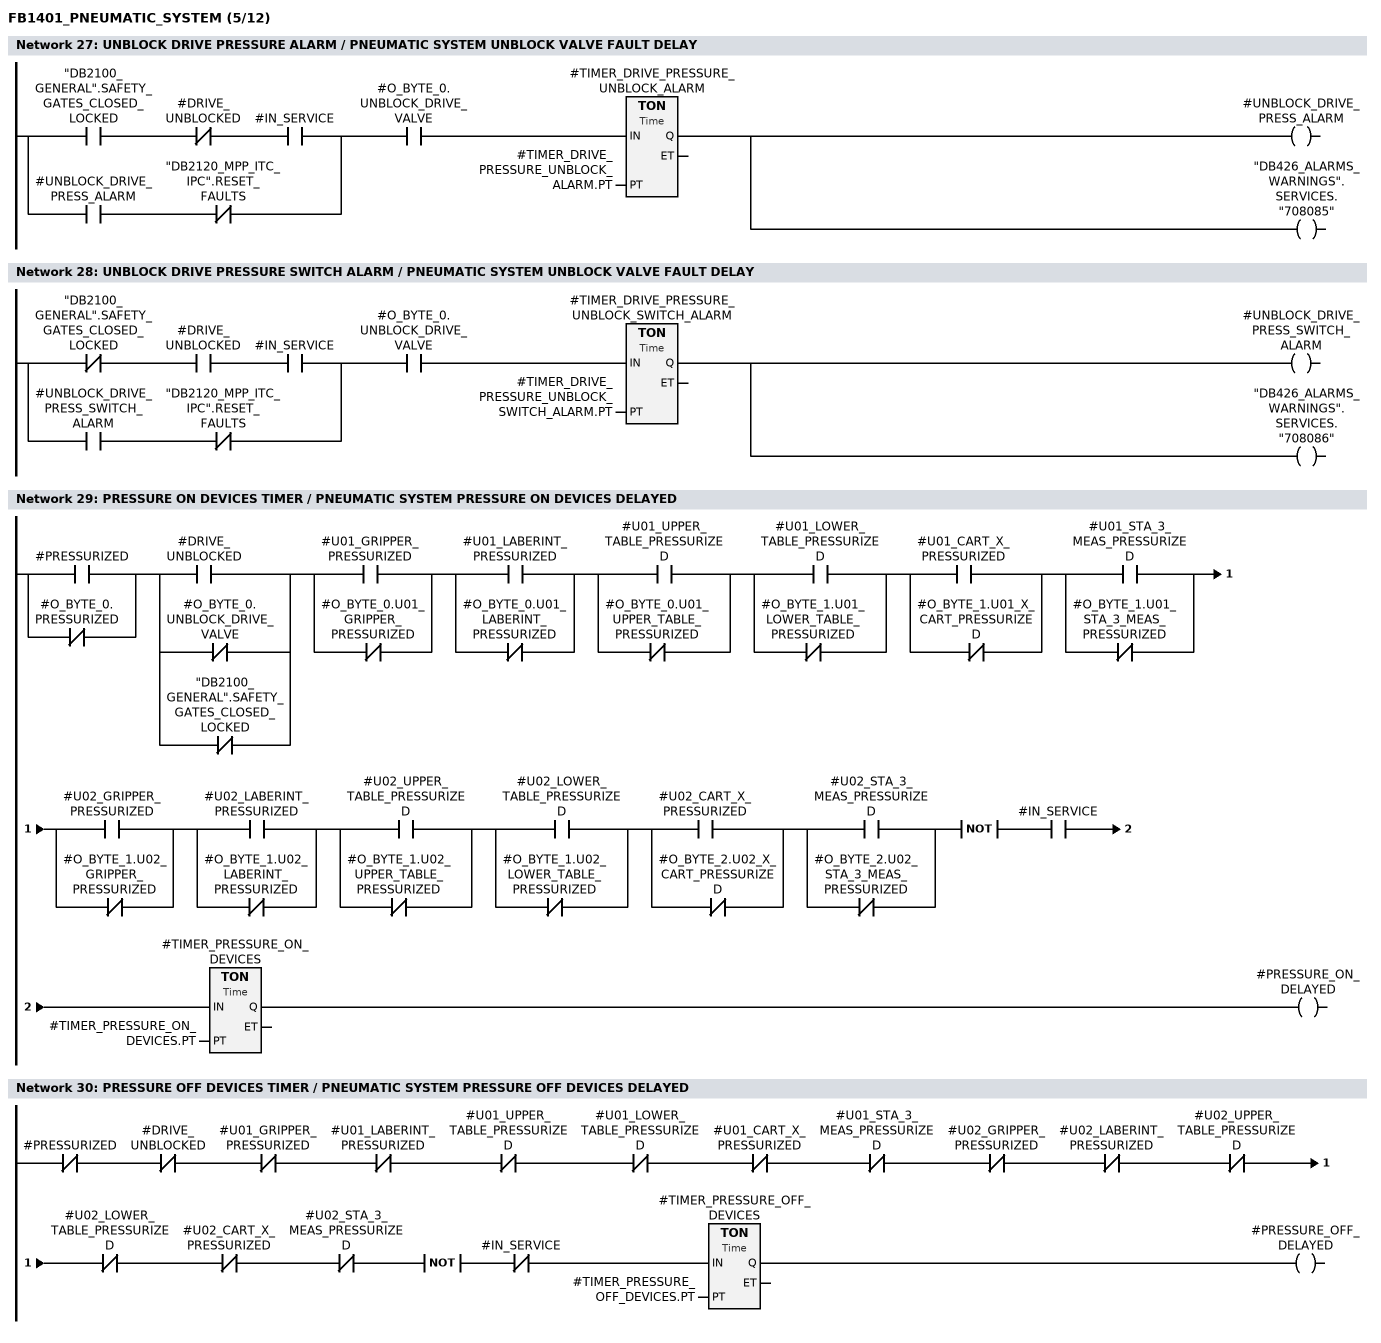
   RUNG wire#powerrail
      Contact( "DB2100_GENERAL".SAFETY_GATES_CLOSED_LOCKED )
      I_Contact( #DRIVE_UNBLOCKED )
      Contact( #IN_SERVICE )
      wire#w1
      Contact( #O_BYTE_0.UNBLOCK_DRIVE_VALVE )
      { S7_Templates := "time_type := Time" } #TIMER_DRIVE_PRESSURE_UNBLOCK_ALARM.TON(pt := #TIMER_DRIVE_PRESSURE_UNBLOCK_ALARM.PT, et =>)
      wire#w2
      Coil( #UNBLOCK_DRIVE_PRESS_ALARM )
   END_RUNG
   RUNG wire#powerrail
      Contact( #UNBLOCK_DRIVE_PRESS_ALARM )
      I_Contact( "DB2120_MPP_ITC_IPC".RESET_FAULTS )
   END_RUNG wire#w1
   RUNG wire#w2
      Coil( "DB426_ALARMS_WARNINGS".SERVICES."708085" )
   END_RUNG
   // the same network as SCL:
   #TIMER_DRIVE_PRESSURE_UNBLOCK_ALARM(IN := (("DB2100_GENERAL".SAFETY_GATES_CLOSED_LOCKED AND NOT #DRIVE_UNBLOCKED AND #IN_SERVICE) OR (#UNBLOCK_DRIVE_PRESS_ALARM AND NOT "DB2120_MPP_ITC_IPC".RESET_FAULTS)) AND #O_BYTE_0.UNBLOCK_DRIVE_VALVE,   // TON
                           PT := #TIMER_DRIVE_PRESSURE_UNBLOCK_ALARM.PT);
   #UNBLOCK_DRIVE_PRESS_ALARM := #TIMER_DRIVE_PRESSURE_UNBLOCK_ALARM.Q;
   "DB426_ALARMS_WARNINGS".SERVICES."708085" := #TIMER_DRIVE_PRESSURE_UNBLOCK_ALARM.Q;
END_REGION

REGION Network 28: UNBLOCK DRIVE PRESSURE SWITCH ALARM / PNEUMATIC SYSTEM UNBLOCK VALVE FAULT DELAY
   RUNG wire#powerrail
      I_Contact( "DB2100_GENERAL".SAFETY_GATES_CLOSED_LOCKED )
      Contact( #DRIVE_UNBLOCKED )
      Contact( #IN_SERVICE )
      wire#w1
      Contact( #O_BYTE_0.UNBLOCK_DRIVE_VALVE )
      { S7_Templates := "time_type := Time" } #TIMER_DRIVE_PRESSURE_UNBLOCK_SWITCH_ALARM.TON(pt := #TIMER_DRIVE_PRESSURE_UNBLOCK_SWITCH_ALARM.PT, et =>)
      wire#w2
      Coil( #UNBLOCK_DRIVE_PRESS_SWITCH_ALARM )
   END_RUNG
   RUNG wire#powerrail
      Contact( #UNBLOCK_DRIVE_PRESS_SWITCH_ALARM )
      I_Contact( "DB2120_MPP_ITC_IPC".RESET_FAULTS )
   END_RUNG wire#w1
   RUNG wire#w2
      Coil( "DB426_ALARMS_WARNINGS".SERVICES."708086" )
   END_RUNG
   // the same network as SCL:
   #TIMER_DRIVE_PRESSURE_UNBLOCK_SWITCH_ALARM(IN := ((NOT "DB2100_GENERAL".SAFETY_GATES_CLOSED_LOCKED AND #DRIVE_UNBLOCKED AND #IN_SERVICE) OR (#UNBLOCK_DRIVE_PRESS_SWITCH_ALARM AND NOT "DB2120_MPP_ITC_IPC".RESET_FAULTS)) AND #O_BYTE_0.UNBLOCK_DRIVE_VALVE,   // TON
                           PT := #TIMER_DRIVE_PRESSURE_UNBLOCK_SWITCH_ALARM.PT);
   #UNBLOCK_DRIVE_PRESS_SWITCH_ALARM := #TIMER_DRIVE_PRESSURE_UNBLOCK_SWITCH_ALARM.Q;
   "DB426_ALARMS_WARNINGS".SERVICES."708086" := #TIMER_DRIVE_PRESSURE_UNBLOCK_SWITCH_ALARM.Q;
END_REGION

REGION Network 29: PRESSURE ON DEVICES TIMER / PNEUMATIC SYSTEM PRESSURE ON DEVICES DELAYED
   RUNG wire#powerrail
      Contact( #PRESSURIZED )
      wire#w1
      Contact( #DRIVE_UNBLOCKED )
      wire#w2
      Contact( #U01_GRIPPER_PRESSURIZED )
      wire#w3
      Contact( #U01_LABERINT_PRESSURIZED )
      wire#w4
      Contact( #U01_UPPER_TABLE_PRESSURIZED )
      wire#w5
      Contact( #U01_LOWER_TABLE_PRESSURIZED )
      wire#w6
      Contact( #U01_CART_X_PRESSURIZED )
      wire#w7
      Contact( #U01_STA_3_MEAS_PRESSURIZED )
      wire#w8
      Contact( #U02_GRIPPER_PRESSURIZED )
      wire#w9
      Contact( #U02_LABERINT_PRESSURIZED )
      wire#w10
      Contact( #U02_UPPER_TABLE_PRESSURIZED )
      wire#w11
      Contact( #U02_LOWER_TABLE_PRESSURIZED )
      wire#w12
      Contact( #U02_CART_X_PRESSURIZED )
      wire#w13
      Contact( #U02_STA_3_MEAS_PRESSURIZED )
      wire#w14
      Not()
      Contact( #IN_SERVICE )
      { S7_Templates := "time_type := Time" } #TIMER_PRESSURE_ON_DEVICES.TON(pt := #TIMER_PRESSURE_ON_DEVICES.PT, et =>)
      Coil( #PRESSURE_ON_DELAYED )
   END_RUNG
   RUNG wire#powerrail
      I_Contact( #O_BYTE_0.PRESSURIZED )
   END_RUNG wire#w1
   RUNG wire#w1
      I_Contact( #O_BYTE_0.UNBLOCK_DRIVE_VALVE )
   END_RUNG wire#w2
   RUNG wire#w1
      I_Contact( "DB2100_GENERAL".SAFETY_GATES_CLOSED_LOCKED )
   END_RUNG wire#w2
   RUNG wire#w2
      I_Contact( #O_BYTE_0.U01_GRIPPER_PRESSURIZED )
   END_RUNG wire#w3
   RUNG wire#w3
      I_Contact( #O_BYTE_0.U01_LABERINT_PRESSURIZED )
   END_RUNG wire#w4
   RUNG wire#w4
      I_Contact( #O_BYTE_0.U01_UPPER_TABLE_PRESSURIZED )
   END_RUNG wire#w5
   RUNG wire#w5
      I_Contact( #O_BYTE_1.U01_LOWER_TABLE_PRESSURIZED )
   END_RUNG wire#w6
   RUNG wire#w6
      I_Contact( #O_BYTE_1.U01_X_CART_PRESSURIZED )
   END_RUNG wire#w7
   RUNG wire#w7
      I_Contact( #O_BYTE_1.U01_STA_3_MEAS_PRESSURIZED )
   END_RUNG wire#w8
   RUNG wire#w8
      I_Contact( #O_BYTE_1.U02_GRIPPER_PRESSURIZED )
   END_RUNG wire#w9
   RUNG wire#w9
      I_Contact( #O_BYTE_1.U02_LABERINT_PRESSURIZED )
   END_RUNG wire#w10
   RUNG wire#w10
      I_Contact( #O_BYTE_1.U02_UPPER_TABLE_PRESSURIZED )
   END_RUNG wire#w11
   RUNG wire#w11
      I_Contact( #O_BYTE_1.U02_LOWER_TABLE_PRESSURIZED )
   END_RUNG wire#w12
   RUNG wire#w12
      I_Contact( #O_BYTE_2.U02_X_CART_PRESSURIZED )
   END_RUNG wire#w13
   RUNG wire#w13
      I_Contact( #O_BYTE_2.U02_STA_3_MEAS_PRESSURIZED )
   END_RUNG wire#w14
   // the same network as SCL:
   #TIMER_PRESSURE_ON_DEVICES(IN := NOT ((#PRESSURIZED OR NOT #O_BYTE_0.PRESSURIZED) AND (#DRIVE_UNBLOCKED OR NOT #O_BYTE_0.UNBLOCK_DRIVE_VALVE OR NOT "DB2100_GENERAL".SAFETY_GATES_CLOSED_LOCKED) AND (#U01_GRIPPER_PRESSURIZED OR NOT #O_BYTE_0.U01_GRIPPER_PRESSURIZED) AND (#U01_LABERINT_PRESSURIZED OR NOT #O_BYTE_0.U01_LABERINT_PRESSURIZED) AND (#U01_UPPER_TABLE_PRESSURIZED OR NOT #O_BYTE_0.U01_UPPER_TABLE_PRESSURIZED) AND (#U01_LOWER_TABLE_PRESSURIZED OR NOT #O_BYTE_1.U01_LOWER_TABLE_PRESSURIZED) AND (#U01_CART_X_PRESSURIZED OR NOT #O_BYTE_1.U01_X_CART_PRESSURIZED) AND (#U01_STA_3_MEAS_PRESSURIZED OR NOT #O_BYTE_1.U01_STA_3_MEAS_PRESSURIZED) AND (#U02_GRIPPER_PRESSURIZED OR NOT #O_BYTE_1.U02_GRIPPER_PRESSURIZED) AND (#U02_LABERINT_PRESSURIZED OR NOT #O_BYTE_1.U02_LABERINT_PRESSURIZED) AND (#U02_UPPER_TABLE_PRESSURIZED OR NOT #O_BYTE_1.U02_UPPER_TABLE_PRESSURIZED) AND (#U02_LOWER_TABLE_PRESSURIZED OR NOT #O_BYTE_1.U02_LOWER_TABLE_PRESSURIZED) AND (#U02_CART_X_PRESSURIZED OR NOT #O_BYTE_2.U02_X_CART_PRESSURIZED) AND (#U02_STA_3_MEAS_PRESSURIZED OR NOT #O_BYTE_2.U02_STA_3_MEAS_PRESSURIZED)) AND #IN_SERVICE,   // TON
                           PT := #TIMER_PRESSURE_ON_DEVICES.PT);
   #PRESSURE_ON_DELAYED := #TIMER_PRESSURE_ON_DEVICES.Q;
END_REGION

REGION Network 30: PRESSURE OFF DEVICES TIMER / PNEUMATIC SYSTEM PRESSURE OFF DEVICES DELAYED
   RUNG wire#powerrail
      I_Contact( #PRESSURIZED )
      I_Contact( #DRIVE_UNBLOCKED )
      I_Contact( #U01_GRIPPER_PRESSURIZED )
      I_Contact( #U01_LABERINT_PRESSURIZED )
      I_Contact( #U01_UPPER_TABLE_PRESSURIZED )
      I_Contact( #U01_LOWER_TABLE_PRESSURIZED )
      I_Contact( #U01_CART_X_PRESSURIZED )
      I_Contact( #U01_STA_3_MEAS_PRESSURIZED )
      I_Contact( #U02_GRIPPER_PRESSURIZED )
      I_Contact( #U02_LABERINT_PRESSURIZED )
      I_Contact( #U02_UPPER_TABLE_PRESSURIZED )
      I_Contact( #U02_LOWER_TABLE_PRESSURIZED )
      I_Contact( #U02_CART_X_PRESSURIZED )
      I_Contact( #U02_STA_3_MEAS_PRESSURIZED )
      Not()
      I_Contact( #IN_SERVICE )
      { S7_Templates := "time_type := Time" } #TIMER_PRESSURE_OFF_DEVICES.TON(pt := #TIMER_PRESSURE_OFF_DEVICES.PT, et =>)
      Coil( #PRESSURE_OFF_DELAYED )
   END_RUNG
   // the same network as SCL:
   #TIMER_PRESSURE_OFF_DEVICES(IN := NOT (NOT #PRESSURIZED AND NOT #DRIVE_UNBLOCKED AND NOT #U01_GRIPPER_PRESSURIZED AND NOT #U01_LABERINT_PRESSURIZED AND NOT #U01_UPPER_TABLE_PRESSURIZED AND NOT #U01_LOWER_TABLE_PRESSURIZED AND NOT #U01_CART_X_PRESSURIZED AND NOT #U01_STA_3_MEAS_PRESSURIZED AND NOT #U02_GRIPPER_PRESSURIZED AND NOT #U02_LABERINT_PRESSURIZED AND NOT #U02_UPPER_TABLE_PRESSURIZED AND NOT #U02_LOWER_TABLE_PRESSURIZED AND NOT #U02_CART_X_PRESSURIZED AND NOT #U02_STA_3_MEAS_PRESSURIZED) AND NOT #IN_SERVICE,   // TON
                           PT := #TIMER_PRESSURE_OFF_DEVICES.PT);
   #PRESSURE_OFF_DELAYED := #TIMER_PRESSURE_OFF_DEVICES.Q;
END_REGION

REGION Network 31: PRESSURIZATION ALARM
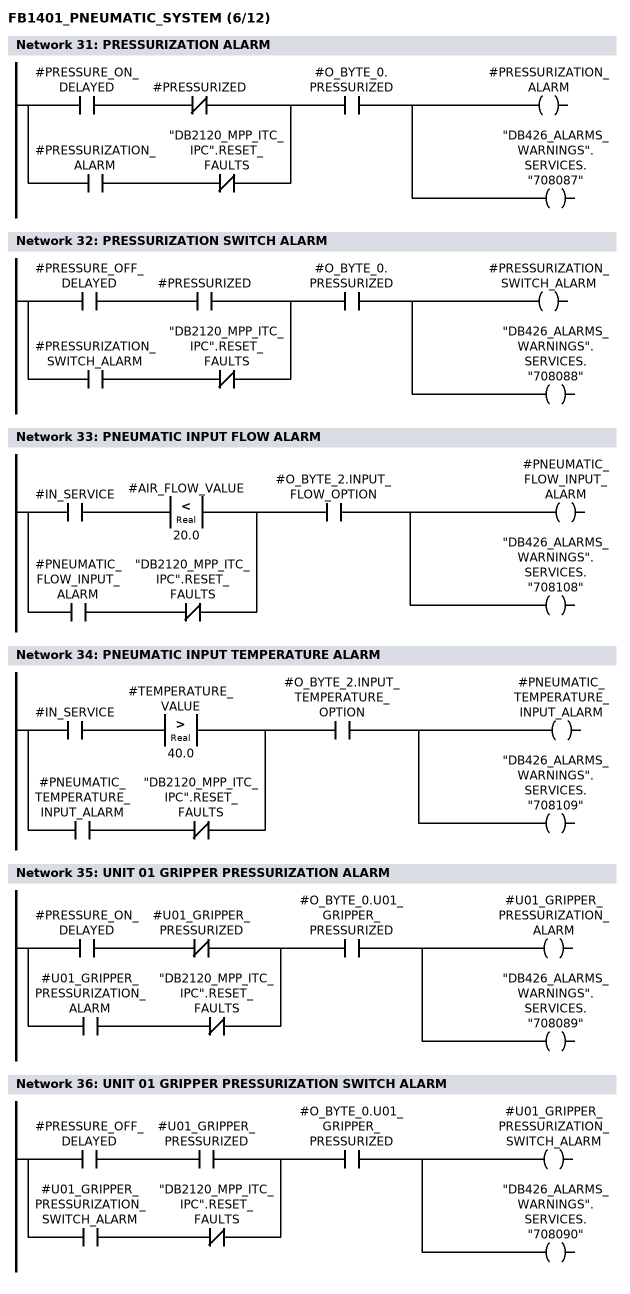
   RUNG wire#powerrail
      Contact( #PRESSURE_ON_DELAYED )
      I_Contact( #PRESSURIZED )
      wire#w1
      Contact( #O_BYTE_0.PRESSURIZED )
      wire#w2
      Coil( #PRESSURIZATION_ALARM )
   END_RUNG
   RUNG wire#powerrail
      Contact( #PRESSURIZATION_ALARM )
      I_Contact( "DB2120_MPP_ITC_IPC".RESET_FAULTS )
   END_RUNG wire#w1
   RUNG wire#w2
      Coil( "DB426_ALARMS_WARNINGS".SERVICES."708087" )
   END_RUNG
   // the same network as SCL:
   #PRESSURIZATION_ALARM := ((#PRESSURE_ON_DELAYED AND NOT #PRESSURIZED) OR (#PRESSURIZATION_ALARM AND NOT "DB2120_MPP_ITC_IPC".RESET_FAULTS)) AND #O_BYTE_0.PRESSURIZED;
   "DB426_ALARMS_WARNINGS".SERVICES."708087" := #PRESSURIZATION_ALARM;
END_REGION

REGION Network 32: PRESSURIZATION SWITCH ALARM
   RUNG wire#powerrail
      Contact( #PRESSURE_OFF_DELAYED )
      Contact( #PRESSURIZED )
      wire#w1
      Contact( #O_BYTE_0.PRESSURIZED )
      wire#w2
      Coil( #PRESSURIZATION_SWITCH_ALARM )
   END_RUNG
   RUNG wire#powerrail
      Contact( #PRESSURIZATION_SWITCH_ALARM )
      I_Contact( "DB2120_MPP_ITC_IPC".RESET_FAULTS )
   END_RUNG wire#w1
   RUNG wire#w2
      Coil( "DB426_ALARMS_WARNINGS".SERVICES."708088" )
   END_RUNG
   // the same network as SCL:
   #PRESSURIZATION_SWITCH_ALARM := ((#PRESSURE_OFF_DELAYED AND #PRESSURIZED) OR (#PRESSURIZATION_SWITCH_ALARM AND NOT "DB2120_MPP_ITC_IPC".RESET_FAULTS)) AND #O_BYTE_0.PRESSURIZED;
   "DB426_ALARMS_WARNINGS".SERVICES."708088" := #PRESSURIZATION_SWITCH_ALARM;
END_REGION

REGION Network 33: PNEUMATIC INPUT FLOW ALARM
   RUNG wire#powerrail
      Contact( #IN_SERVICE )
      { S7_Templates := "SrcType := Real" } LT_Contact(in1 := #AIR_FLOW_VALUE, in2 := 20.0)
      wire#w1
      Contact( #O_BYTE_2.INPUT_FLOW_OPTION )
      wire#w2
      Coil( #PNEUMATIC_FLOW_INPUT_ALARM )
   END_RUNG
   RUNG wire#powerrail
      Contact( #PNEUMATIC_FLOW_INPUT_ALARM )
      I_Contact( "DB2120_MPP_ITC_IPC".RESET_FAULTS )
   END_RUNG wire#w1
   RUNG wire#w2
      Coil( "DB426_ALARMS_WARNINGS".SERVICES."708108" )
   END_RUNG
   // the same network as SCL:
   #PNEUMATIC_FLOW_INPUT_ALARM := ((#IN_SERVICE AND (#AIR_FLOW_VALUE < 20.0)) OR (#PNEUMATIC_FLOW_INPUT_ALARM AND NOT "DB2120_MPP_ITC_IPC".RESET_FAULTS)) AND #O_BYTE_2.INPUT_FLOW_OPTION;
   "DB426_ALARMS_WARNINGS".SERVICES."708108" := #PNEUMATIC_FLOW_INPUT_ALARM;
END_REGION

REGION Network 34: PNEUMATIC INPUT TEMPERATURE ALARM
   RUNG wire#powerrail
      Contact( #IN_SERVICE )
      { S7_Templates := "SrcType := Real" } GT_Contact(in1 := #TEMPERATURE_VALUE, in2 := 40.0)
      wire#w1
      Contact( #O_BYTE_2.INPUT_TEMPERATURE_OPTION )
      wire#w2
      Coil( #PNEUMATIC_TEMPERATURE_INPUT_ALARM )
   END_RUNG
   RUNG wire#powerrail
      Contact( #PNEUMATIC_TEMPERATURE_INPUT_ALARM )
      I_Contact( "DB2120_MPP_ITC_IPC".RESET_FAULTS )
   END_RUNG wire#w1
   RUNG wire#w2
      Coil( "DB426_ALARMS_WARNINGS".SERVICES."708109" )
   END_RUNG
   // the same network as SCL:
   #PNEUMATIC_TEMPERATURE_INPUT_ALARM := ((#IN_SERVICE AND (#TEMPERATURE_VALUE > 40.0)) OR (#PNEUMATIC_TEMPERATURE_INPUT_ALARM AND NOT "DB2120_MPP_ITC_IPC".RESET_FAULTS)) AND #O_BYTE_2.INPUT_TEMPERATURE_OPTION;
   "DB426_ALARMS_WARNINGS".SERVICES."708109" := #PNEUMATIC_TEMPERATURE_INPUT_ALARM;
END_REGION

REGION Network 35: UNIT 01 GRIPPER PRESSURIZATION ALARM
   RUNG wire#powerrail
      Contact( #PRESSURE_ON_DELAYED )
      I_Contact( #U01_GRIPPER_PRESSURIZED )
      wire#w1
      Contact( #O_BYTE_0.U01_GRIPPER_PRESSURIZED )
      wire#w2
      Coil( #U01_GRIPPER_PRESSURIZATION_ALARM )
   END_RUNG
   RUNG wire#powerrail
      Contact( #U01_GRIPPER_PRESSURIZATION_ALARM )
      I_Contact( "DB2120_MPP_ITC_IPC".RESET_FAULTS )
   END_RUNG wire#w1
   RUNG wire#w2
      Coil( "DB426_ALARMS_WARNINGS".SERVICES."708089" )
   END_RUNG
   // the same network as SCL:
   #U01_GRIPPER_PRESSURIZATION_ALARM := ((#PRESSURE_ON_DELAYED AND NOT #U01_GRIPPER_PRESSURIZED) OR (#U01_GRIPPER_PRESSURIZATION_ALARM AND NOT "DB2120_MPP_ITC_IPC".RESET_FAULTS)) AND #O_BYTE_0.U01_GRIPPER_PRESSURIZED;
   "DB426_ALARMS_WARNINGS".SERVICES."708089" := #U01_GRIPPER_PRESSURIZATION_ALARM;
END_REGION

REGION Network 36: UNIT 01 GRIPPER PRESSURIZATION SWITCH ALARM
   RUNG wire#powerrail
      Contact( #PRESSURE_OFF_DELAYED )
      Contact( #U01_GRIPPER_PRESSURIZED )
      wire#w1
      Contact( #O_BYTE_0.U01_GRIPPER_PRESSURIZED )
      wire#w2
      Coil( #U01_GRIPPER_PRESSURIZATION_SWITCH_ALARM )
   END_RUNG
   RUNG wire#powerrail
      Contact( #U01_GRIPPER_PRESSURIZATION_SWITCH_ALARM )
      I_Contact( "DB2120_MPP_ITC_IPC".RESET_FAULTS )
   END_RUNG wire#w1
   RUNG wire#w2
      Coil( "DB426_ALARMS_WARNINGS".SERVICES."708090" )
   END_RUNG
   // the same network as SCL:
   #U01_GRIPPER_PRESSURIZATION_SWITCH_ALARM := ((#PRESSURE_OFF_DELAYED AND #U01_GRIPPER_PRESSURIZED) OR (#U01_GRIPPER_PRESSURIZATION_SWITCH_ALARM AND NOT "DB2120_MPP_ITC_IPC".RESET_FAULTS)) AND #O_BYTE_0.U01_GRIPPER_PRESSURIZED;
   "DB426_ALARMS_WARNINGS".SERVICES."708090" := #U01_GRIPPER_PRESSURIZATION_SWITCH_ALARM;
END_REGION

REGION Network 37: UNIT 01 LABERINT PRESSURIZATION ALARM
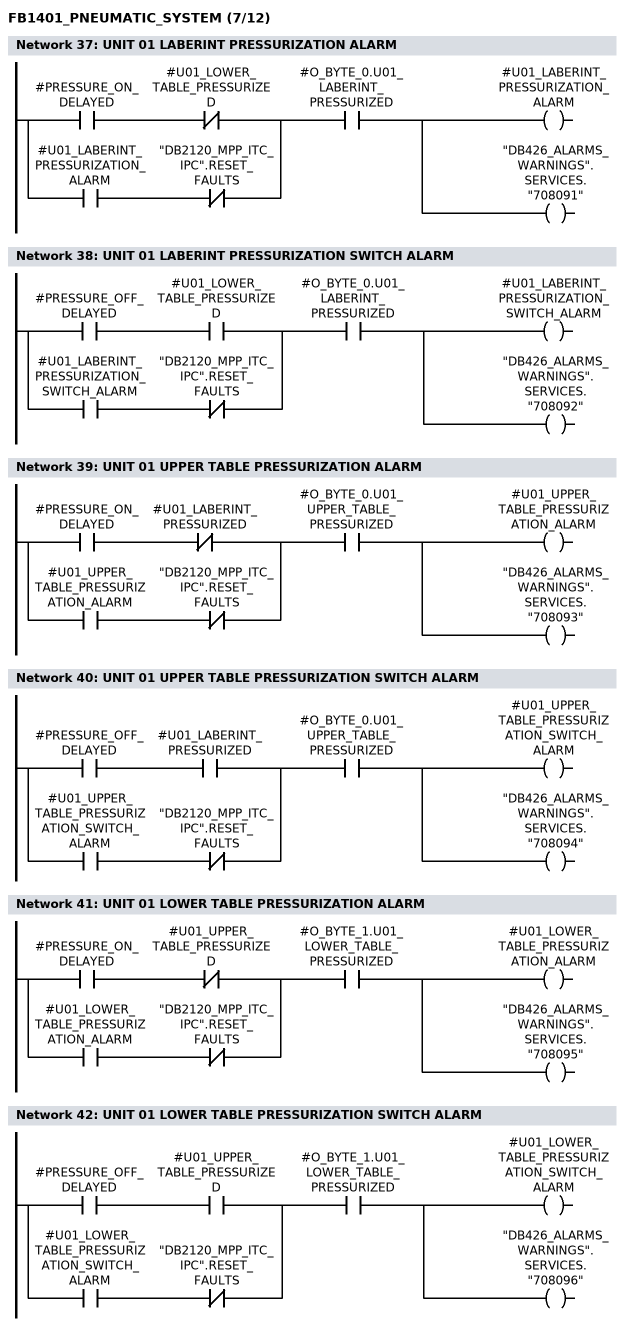
   RUNG wire#powerrail
      Contact( #PRESSURE_ON_DELAYED )
      I_Contact( #U01_LOWER_TABLE_PRESSURIZED )
      wire#w1
      Contact( #O_BYTE_0.U01_LABERINT_PRESSURIZED )
      wire#w2
      Coil( #U01_LABERINT_PRESSURIZATION_ALARM )
   END_RUNG
   RUNG wire#powerrail
      Contact( #U01_LABERINT_PRESSURIZATION_ALARM )
      I_Contact( "DB2120_MPP_ITC_IPC".RESET_FAULTS )
   END_RUNG wire#w1
   RUNG wire#w2
      Coil( "DB426_ALARMS_WARNINGS".SERVICES."708091" )
   END_RUNG
   // the same network as SCL:
   #U01_LABERINT_PRESSURIZATION_ALARM := ((#PRESSURE_ON_DELAYED AND NOT #U01_LOWER_TABLE_PRESSURIZED) OR (#U01_LABERINT_PRESSURIZATION_ALARM AND NOT "DB2120_MPP_ITC_IPC".RESET_FAULTS)) AND #O_BYTE_0.U01_LABERINT_PRESSURIZED;
   "DB426_ALARMS_WARNINGS".SERVICES."708091" := #U01_LABERINT_PRESSURIZATION_ALARM;
END_REGION

REGION Network 38: UNIT 01 LABERINT PRESSURIZATION SWITCH ALARM
   RUNG wire#powerrail
      Contact( #PRESSURE_OFF_DELAYED )
      Contact( #U01_LOWER_TABLE_PRESSURIZED )
      wire#w1
      Contact( #O_BYTE_0.U01_LABERINT_PRESSURIZED )
      wire#w2
      Coil( #U01_LABERINT_PRESSURIZATION_SWITCH_ALARM )
   END_RUNG
   RUNG wire#powerrail
      Contact( #U01_LABERINT_PRESSURIZATION_SWITCH_ALARM )
      I_Contact( "DB2120_MPP_ITC_IPC".RESET_FAULTS )
   END_RUNG wire#w1
   RUNG wire#w2
      Coil( "DB426_ALARMS_WARNINGS".SERVICES."708092" )
   END_RUNG
   // the same network as SCL:
   #U01_LABERINT_PRESSURIZATION_SWITCH_ALARM := ((#PRESSURE_OFF_DELAYED AND #U01_LOWER_TABLE_PRESSURIZED) OR (#U01_LABERINT_PRESSURIZATION_SWITCH_ALARM AND NOT "DB2120_MPP_ITC_IPC".RESET_FAULTS)) AND #O_BYTE_0.U01_LABERINT_PRESSURIZED;
   "DB426_ALARMS_WARNINGS".SERVICES."708092" := #U01_LABERINT_PRESSURIZATION_SWITCH_ALARM;
END_REGION

REGION Network 39: UNIT 01 UPPER TABLE PRESSURIZATION ALARM
   RUNG wire#powerrail
      Contact( #PRESSURE_ON_DELAYED )
      I_Contact( #U01_LABERINT_PRESSURIZED )
      wire#w1
      Contact( #O_BYTE_0.U01_UPPER_TABLE_PRESSURIZED )
      wire#w2
      Coil( #U01_UPPER_TABLE_PRESSURIZATION_ALARM )
   END_RUNG
   RUNG wire#powerrail
      Contact( #U01_UPPER_TABLE_PRESSURIZATION_ALARM )
      I_Contact( "DB2120_MPP_ITC_IPC".RESET_FAULTS )
   END_RUNG wire#w1
   RUNG wire#w2
      Coil( "DB426_ALARMS_WARNINGS".SERVICES."708093" )
   END_RUNG
   // the same network as SCL:
   #U01_UPPER_TABLE_PRESSURIZATION_ALARM := ((#PRESSURE_ON_DELAYED AND NOT #U01_LABERINT_PRESSURIZED) OR (#U01_UPPER_TABLE_PRESSURIZATION_ALARM AND NOT "DB2120_MPP_ITC_IPC".RESET_FAULTS)) AND #O_BYTE_0.U01_UPPER_TABLE_PRESSURIZED;
   "DB426_ALARMS_WARNINGS".SERVICES."708093" := #U01_UPPER_TABLE_PRESSURIZATION_ALARM;
END_REGION

REGION Network 40: UNIT 01 UPPER TABLE PRESSURIZATION SWITCH ALARM
   RUNG wire#powerrail
      Contact( #PRESSURE_OFF_DELAYED )
      Contact( #U01_LABERINT_PRESSURIZED )
      wire#w1
      Contact( #O_BYTE_0.U01_UPPER_TABLE_PRESSURIZED )
      wire#w2
      Coil( #U01_UPPER_TABLE_PRESSURIZATION_SWITCH_ALARM )
   END_RUNG
   RUNG wire#powerrail
      Contact( #U01_UPPER_TABLE_PRESSURIZATION_SWITCH_ALARM )
      I_Contact( "DB2120_MPP_ITC_IPC".RESET_FAULTS )
   END_RUNG wire#w1
   RUNG wire#w2
      Coil( "DB426_ALARMS_WARNINGS".SERVICES."708094" )
   END_RUNG
   // the same network as SCL:
   #U01_UPPER_TABLE_PRESSURIZATION_SWITCH_ALARM := ((#PRESSURE_OFF_DELAYED AND #U01_LABERINT_PRESSURIZED) OR (#U01_UPPER_TABLE_PRESSURIZATION_SWITCH_ALARM AND NOT "DB2120_MPP_ITC_IPC".RESET_FAULTS)) AND #O_BYTE_0.U01_UPPER_TABLE_PRESSURIZED;
   "DB426_ALARMS_WARNINGS".SERVICES."708094" := #U01_UPPER_TABLE_PRESSURIZATION_SWITCH_ALARM;
END_REGION

REGION Network 41: UNIT 01 LOWER TABLE PRESSURIZATION ALARM
   RUNG wire#powerrail
      Contact( #PRESSURE_ON_DELAYED )
      I_Contact( #U01_UPPER_TABLE_PRESSURIZED )
      wire#w1
      Contact( #O_BYTE_1.U01_LOWER_TABLE_PRESSURIZED )
      wire#w2
      Coil( #U01_LOWER_TABLE_PRESSURIZATION_ALARM )
   END_RUNG
   RUNG wire#powerrail
      Contact( #U01_LOWER_TABLE_PRESSURIZATION_ALARM )
      I_Contact( "DB2120_MPP_ITC_IPC".RESET_FAULTS )
   END_RUNG wire#w1
   RUNG wire#w2
      Coil( "DB426_ALARMS_WARNINGS".SERVICES."708095" )
   END_RUNG
   // the same network as SCL:
   #U01_LOWER_TABLE_PRESSURIZATION_ALARM := ((#PRESSURE_ON_DELAYED AND NOT #U01_UPPER_TABLE_PRESSURIZED) OR (#U01_LOWER_TABLE_PRESSURIZATION_ALARM AND NOT "DB2120_MPP_ITC_IPC".RESET_FAULTS)) AND #O_BYTE_1.U01_LOWER_TABLE_PRESSURIZED;
   "DB426_ALARMS_WARNINGS".SERVICES."708095" := #U01_LOWER_TABLE_PRESSURIZATION_ALARM;
END_REGION

REGION Network 42: UNIT 01 LOWER TABLE PRESSURIZATION SWITCH ALARM
   RUNG wire#powerrail
      Contact( #PRESSURE_OFF_DELAYED )
      Contact( #U01_UPPER_TABLE_PRESSURIZED )
      wire#w1
      Contact( #O_BYTE_1.U01_LOWER_TABLE_PRESSURIZED )
      wire#w2
      Coil( #U01_LOWER_TABLE_PRESSURIZATION_SWITCH_ALARM )
   END_RUNG
   RUNG wire#powerrail
      Contact( #U01_LOWER_TABLE_PRESSURIZATION_SWITCH_ALARM )
      I_Contact( "DB2120_MPP_ITC_IPC".RESET_FAULTS )
   END_RUNG wire#w1
   RUNG wire#w2
      Coil( "DB426_ALARMS_WARNINGS".SERVICES."708096" )
   END_RUNG
   // the same network as SCL:
   #U01_LOWER_TABLE_PRESSURIZATION_SWITCH_ALARM := ((#PRESSURE_OFF_DELAYED AND #U01_UPPER_TABLE_PRESSURIZED) OR (#U01_LOWER_TABLE_PRESSURIZATION_SWITCH_ALARM AND NOT "DB2120_MPP_ITC_IPC".RESET_FAULTS)) AND #O_BYTE_1.U01_LOWER_TABLE_PRESSURIZED;
   "DB426_ALARMS_WARNINGS".SERVICES."708096" := #U01_LOWER_TABLE_PRESSURIZATION_SWITCH_ALARM;
END_REGION

REGION Network 43: UNIT 01 CART AXIS X PRESSURIZATION ALARM
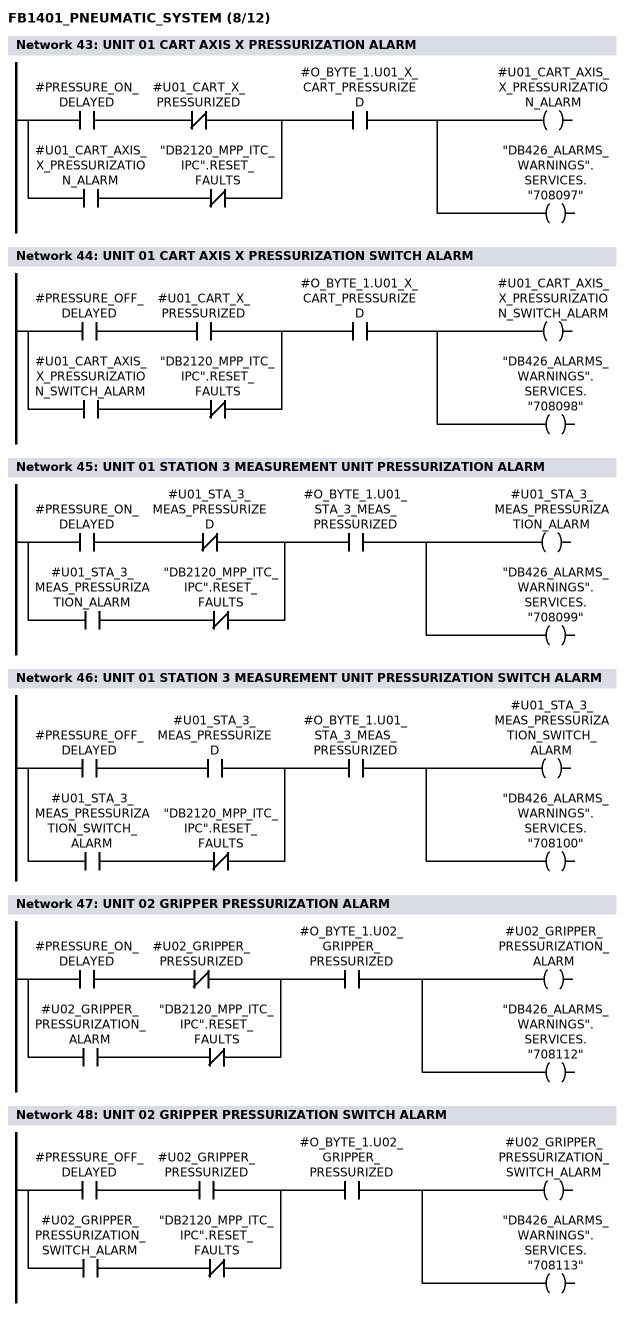
   RUNG wire#powerrail
      Contact( #PRESSURE_ON_DELAYED )
      I_Contact( #U01_CART_X_PRESSURIZED )
      wire#w1
      Contact( #O_BYTE_1.U01_X_CART_PRESSURIZED )
      wire#w2
      Coil( #U01_CART_AXIS_X_PRESSURIZATION_ALARM )
   END_RUNG
   RUNG wire#powerrail
      Contact( #U01_CART_AXIS_X_PRESSURIZATION_ALARM )
      I_Contact( "DB2120_MPP_ITC_IPC".RESET_FAULTS )
   END_RUNG wire#w1
   RUNG wire#w2
      Coil( "DB426_ALARMS_WARNINGS".SERVICES."708097" )
   END_RUNG
   // the same network as SCL:
   #U01_CART_AXIS_X_PRESSURIZATION_ALARM := ((#PRESSURE_ON_DELAYED AND NOT #U01_CART_X_PRESSURIZED) OR (#U01_CART_AXIS_X_PRESSURIZATION_ALARM AND NOT "DB2120_MPP_ITC_IPC".RESET_FAULTS)) AND #O_BYTE_1.U01_X_CART_PRESSURIZED;
   "DB426_ALARMS_WARNINGS".SERVICES."708097" := #U01_CART_AXIS_X_PRESSURIZATION_ALARM;
END_REGION

REGION Network 44: UNIT 01 CART AXIS X PRESSURIZATION SWITCH ALARM
   RUNG wire#powerrail
      Contact( #PRESSURE_OFF_DELAYED )
      Contact( #U01_CART_X_PRESSURIZED )
      wire#w1
      Contact( #O_BYTE_1.U01_X_CART_PRESSURIZED )
      wire#w2
      Coil( #U01_CART_AXIS_X_PRESSURIZATION_SWITCH_ALARM )
   END_RUNG
   RUNG wire#powerrail
      Contact( #U01_CART_AXIS_X_PRESSURIZATION_SWITCH_ALARM )
      I_Contact( "DB2120_MPP_ITC_IPC".RESET_FAULTS )
   END_RUNG wire#w1
   RUNG wire#w2
      Coil( "DB426_ALARMS_WARNINGS".SERVICES."708098" )
   END_RUNG
   // the same network as SCL:
   #U01_CART_AXIS_X_PRESSURIZATION_SWITCH_ALARM := ((#PRESSURE_OFF_DELAYED AND #U01_CART_X_PRESSURIZED) OR (#U01_CART_AXIS_X_PRESSURIZATION_SWITCH_ALARM AND NOT "DB2120_MPP_ITC_IPC".RESET_FAULTS)) AND #O_BYTE_1.U01_X_CART_PRESSURIZED;
   "DB426_ALARMS_WARNINGS".SERVICES."708098" := #U01_CART_AXIS_X_PRESSURIZATION_SWITCH_ALARM;
END_REGION

REGION Network 45: UNIT 01 STATION 3 MEASUREMENT UNIT PRESSURIZATION ALARM
   RUNG wire#powerrail
      Contact( #PRESSURE_ON_DELAYED )
      I_Contact( #U01_STA_3_MEAS_PRESSURIZED )
      wire#w1
      Contact( #O_BYTE_1.U01_STA_3_MEAS_PRESSURIZED )
      wire#w2
      Coil( #U01_STA_3_MEAS_PRESSURIZATION_ALARM )
   END_RUNG
   RUNG wire#powerrail
      Contact( #U01_STA_3_MEAS_PRESSURIZATION_ALARM )
      I_Contact( "DB2120_MPP_ITC_IPC".RESET_FAULTS )
   END_RUNG wire#w1
   RUNG wire#w2
      Coil( "DB426_ALARMS_WARNINGS".SERVICES."708099" )
   END_RUNG
   // the same network as SCL:
   #U01_STA_3_MEAS_PRESSURIZATION_ALARM := ((#PRESSURE_ON_DELAYED AND NOT #U01_STA_3_MEAS_PRESSURIZED) OR (#U01_STA_3_MEAS_PRESSURIZATION_ALARM AND NOT "DB2120_MPP_ITC_IPC".RESET_FAULTS)) AND #O_BYTE_1.U01_STA_3_MEAS_PRESSURIZED;
   "DB426_ALARMS_WARNINGS".SERVICES."708099" := #U01_STA_3_MEAS_PRESSURIZATION_ALARM;
END_REGION

REGION Network 46: UNIT 01 STATION 3 MEASUREMENT UNIT PRESSURIZATION SWITCH ALARM
   RUNG wire#powerrail
      Contact( #PRESSURE_OFF_DELAYED )
      Contact( #U01_STA_3_MEAS_PRESSURIZED )
      wire#w1
      Contact( #O_BYTE_1.U01_STA_3_MEAS_PRESSURIZED )
      wire#w2
      Coil( #U01_STA_3_MEAS_PRESSURIZATION_SWITCH_ALARM )
   END_RUNG
   RUNG wire#powerrail
      Contact( #U01_STA_3_MEAS_PRESSURIZATION_SWITCH_ALARM )
      I_Contact( "DB2120_MPP_ITC_IPC".RESET_FAULTS )
   END_RUNG wire#w1
   RUNG wire#w2
      Coil( "DB426_ALARMS_WARNINGS".SERVICES."708100" )
   END_RUNG
   // the same network as SCL:
   #U01_STA_3_MEAS_PRESSURIZATION_SWITCH_ALARM := ((#PRESSURE_OFF_DELAYED AND #U01_STA_3_MEAS_PRESSURIZED) OR (#U01_STA_3_MEAS_PRESSURIZATION_SWITCH_ALARM AND NOT "DB2120_MPP_ITC_IPC".RESET_FAULTS)) AND #O_BYTE_1.U01_STA_3_MEAS_PRESSURIZED;
   "DB426_ALARMS_WARNINGS".SERVICES."708100" := #U01_STA_3_MEAS_PRESSURIZATION_SWITCH_ALARM;
END_REGION

REGION Network 47: UNIT 02 GRIPPER PRESSURIZATION ALARM
   RUNG wire#powerrail
      Contact( #PRESSURE_ON_DELAYED )
      I_Contact( #U02_GRIPPER_PRESSURIZED )
      wire#w1
      Contact( #O_BYTE_1.U02_GRIPPER_PRESSURIZED )
      wire#w2
      Coil( #U02_GRIPPER_PRESSURIZATION_ALARM )
   END_RUNG
   RUNG wire#powerrail
      Contact( #U02_GRIPPER_PRESSURIZATION_ALARM )
      I_Contact( "DB2120_MPP_ITC_IPC".RESET_FAULTS )
   END_RUNG wire#w1
   RUNG wire#w2
      Coil( "DB426_ALARMS_WARNINGS".SERVICES."708112" )
   END_RUNG
   // the same network as SCL:
   #U02_GRIPPER_PRESSURIZATION_ALARM := ((#PRESSURE_ON_DELAYED AND NOT #U02_GRIPPER_PRESSURIZED) OR (#U02_GRIPPER_PRESSURIZATION_ALARM AND NOT "DB2120_MPP_ITC_IPC".RESET_FAULTS)) AND #O_BYTE_1.U02_GRIPPER_PRESSURIZED;
   "DB426_ALARMS_WARNINGS".SERVICES."708112" := #U02_GRIPPER_PRESSURIZATION_ALARM;
END_REGION

REGION Network 48: UNIT 02 GRIPPER PRESSURIZATION SWITCH ALARM
   RUNG wire#powerrail
      Contact( #PRESSURE_OFF_DELAYED )
      Contact( #U02_GRIPPER_PRESSURIZED )
      wire#w1
      Contact( #O_BYTE_1.U02_GRIPPER_PRESSURIZED )
      wire#w2
      Coil( #U02_GRIPPER_PRESSURIZATION_SWITCH_ALARM )
   END_RUNG
   RUNG wire#powerrail
      Contact( #U02_GRIPPER_PRESSURIZATION_SWITCH_ALARM )
      I_Contact( "DB2120_MPP_ITC_IPC".RESET_FAULTS )
   END_RUNG wire#w1
   RUNG wire#w2
      Coil( "DB426_ALARMS_WARNINGS".SERVICES."708113" )
   END_RUNG
   // the same network as SCL:
   #U02_GRIPPER_PRESSURIZATION_SWITCH_ALARM := ((#PRESSURE_OFF_DELAYED AND #U02_GRIPPER_PRESSURIZED) OR (#U02_GRIPPER_PRESSURIZATION_SWITCH_ALARM AND NOT "DB2120_MPP_ITC_IPC".RESET_FAULTS)) AND #O_BYTE_1.U02_GRIPPER_PRESSURIZED;
   "DB426_ALARMS_WARNINGS".SERVICES."708113" := #U02_GRIPPER_PRESSURIZATION_SWITCH_ALARM;
END_REGION

REGION Network 49: UNIT 02 LABERINT PRESSURIZATION ALARM
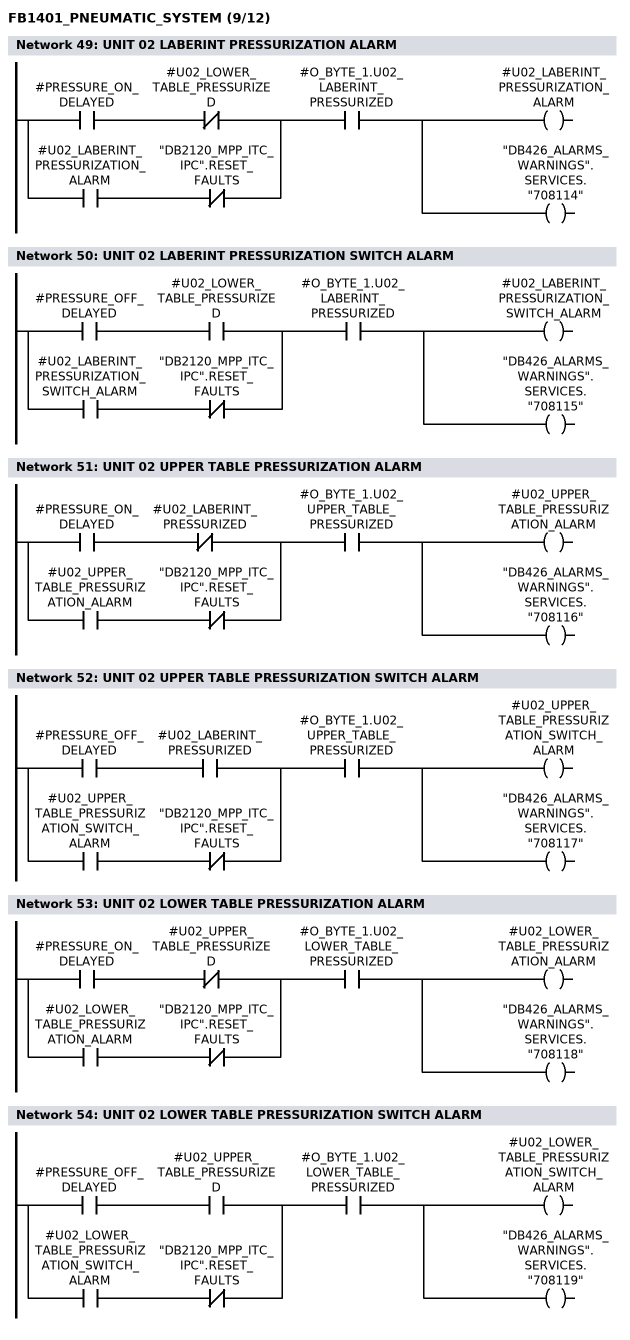
   RUNG wire#powerrail
      Contact( #PRESSURE_ON_DELAYED )
      I_Contact( #U02_LOWER_TABLE_PRESSURIZED )
      wire#w1
      Contact( #O_BYTE_1.U02_LABERINT_PRESSURIZED )
      wire#w2
      Coil( #U02_LABERINT_PRESSURIZATION_ALARM )
   END_RUNG
   RUNG wire#powerrail
      Contact( #U02_LABERINT_PRESSURIZATION_ALARM )
      I_Contact( "DB2120_MPP_ITC_IPC".RESET_FAULTS )
   END_RUNG wire#w1
   RUNG wire#w2
      Coil( "DB426_ALARMS_WARNINGS".SERVICES."708114" )
   END_RUNG
   // the same network as SCL:
   #U02_LABERINT_PRESSURIZATION_ALARM := ((#PRESSURE_ON_DELAYED AND NOT #U02_LOWER_TABLE_PRESSURIZED) OR (#U02_LABERINT_PRESSURIZATION_ALARM AND NOT "DB2120_MPP_ITC_IPC".RESET_FAULTS)) AND #O_BYTE_1.U02_LABERINT_PRESSURIZED;
   "DB426_ALARMS_WARNINGS".SERVICES."708114" := #U02_LABERINT_PRESSURIZATION_ALARM;
END_REGION

REGION Network 50: UNIT 02 LABERINT PRESSURIZATION SWITCH ALARM
   RUNG wire#powerrail
      Contact( #PRESSURE_OFF_DELAYED )
      Contact( #U02_LOWER_TABLE_PRESSURIZED )
      wire#w1
      Contact( #O_BYTE_1.U02_LABERINT_PRESSURIZED )
      wire#w2
      Coil( #U02_LABERINT_PRESSURIZATION_SWITCH_ALARM )
   END_RUNG
   RUNG wire#powerrail
      Contact( #U02_LABERINT_PRESSURIZATION_SWITCH_ALARM )
      I_Contact( "DB2120_MPP_ITC_IPC".RESET_FAULTS )
   END_RUNG wire#w1
   RUNG wire#w2
      Coil( "DB426_ALARMS_WARNINGS".SERVICES."708115" )
   END_RUNG
   // the same network as SCL:
   #U02_LABERINT_PRESSURIZATION_SWITCH_ALARM := ((#PRESSURE_OFF_DELAYED AND #U02_LOWER_TABLE_PRESSURIZED) OR (#U02_LABERINT_PRESSURIZATION_SWITCH_ALARM AND NOT "DB2120_MPP_ITC_IPC".RESET_FAULTS)) AND #O_BYTE_1.U02_LABERINT_PRESSURIZED;
   "DB426_ALARMS_WARNINGS".SERVICES."708115" := #U02_LABERINT_PRESSURIZATION_SWITCH_ALARM;
END_REGION

REGION Network 51: UNIT 02 UPPER TABLE PRESSURIZATION ALARM
   RUNG wire#powerrail
      Contact( #PRESSURE_ON_DELAYED )
      I_Contact( #U02_LABERINT_PRESSURIZED )
      wire#w1
      Contact( #O_BYTE_1.U02_UPPER_TABLE_PRESSURIZED )
      wire#w2
      Coil( #U02_UPPER_TABLE_PRESSURIZATION_ALARM )
   END_RUNG
   RUNG wire#powerrail
      Contact( #U02_UPPER_TABLE_PRESSURIZATION_ALARM )
      I_Contact( "DB2120_MPP_ITC_IPC".RESET_FAULTS )
   END_RUNG wire#w1
   RUNG wire#w2
      Coil( "DB426_ALARMS_WARNINGS".SERVICES."708116" )
   END_RUNG
   // the same network as SCL:
   #U02_UPPER_TABLE_PRESSURIZATION_ALARM := ((#PRESSURE_ON_DELAYED AND NOT #U02_LABERINT_PRESSURIZED) OR (#U02_UPPER_TABLE_PRESSURIZATION_ALARM AND NOT "DB2120_MPP_ITC_IPC".RESET_FAULTS)) AND #O_BYTE_1.U02_UPPER_TABLE_PRESSURIZED;
   "DB426_ALARMS_WARNINGS".SERVICES."708116" := #U02_UPPER_TABLE_PRESSURIZATION_ALARM;
END_REGION

REGION Network 52: UNIT 02 UPPER TABLE PRESSURIZATION SWITCH ALARM
   RUNG wire#powerrail
      Contact( #PRESSURE_OFF_DELAYED )
      Contact( #U02_LABERINT_PRESSURIZED )
      wire#w1
      Contact( #O_BYTE_1.U02_UPPER_TABLE_PRESSURIZED )
      wire#w2
      Coil( #U02_UPPER_TABLE_PRESSURIZATION_SWITCH_ALARM )
   END_RUNG
   RUNG wire#powerrail
      Contact( #U02_UPPER_TABLE_PRESSURIZATION_SWITCH_ALARM )
      I_Contact( "DB2120_MPP_ITC_IPC".RESET_FAULTS )
   END_RUNG wire#w1
   RUNG wire#w2
      Coil( "DB426_ALARMS_WARNINGS".SERVICES."708117" )
   END_RUNG
   // the same network as SCL:
   #U02_UPPER_TABLE_PRESSURIZATION_SWITCH_ALARM := ((#PRESSURE_OFF_DELAYED AND #U02_LABERINT_PRESSURIZED) OR (#U02_UPPER_TABLE_PRESSURIZATION_SWITCH_ALARM AND NOT "DB2120_MPP_ITC_IPC".RESET_FAULTS)) AND #O_BYTE_1.U02_UPPER_TABLE_PRESSURIZED;
   "DB426_ALARMS_WARNINGS".SERVICES."708117" := #U02_UPPER_TABLE_PRESSURIZATION_SWITCH_ALARM;
END_REGION

REGION Network 53: UNIT 02 LOWER TABLE PRESSURIZATION ALARM
   RUNG wire#powerrail
      Contact( #PRESSURE_ON_DELAYED )
      I_Contact( #U02_UPPER_TABLE_PRESSURIZED )
      wire#w1
      Contact( #O_BYTE_1.U02_LOWER_TABLE_PRESSURIZED )
      wire#w2
      Coil( #U02_LOWER_TABLE_PRESSURIZATION_ALARM )
   END_RUNG
   RUNG wire#powerrail
      Contact( #U02_LOWER_TABLE_PRESSURIZATION_ALARM )
      I_Contact( "DB2120_MPP_ITC_IPC".RESET_FAULTS )
   END_RUNG wire#w1
   RUNG wire#w2
      Coil( "DB426_ALARMS_WARNINGS".SERVICES."708118" )
   END_RUNG
   // the same network as SCL:
   #U02_LOWER_TABLE_PRESSURIZATION_ALARM := ((#PRESSURE_ON_DELAYED AND NOT #U02_UPPER_TABLE_PRESSURIZED) OR (#U02_LOWER_TABLE_PRESSURIZATION_ALARM AND NOT "DB2120_MPP_ITC_IPC".RESET_FAULTS)) AND #O_BYTE_1.U02_LOWER_TABLE_PRESSURIZED;
   "DB426_ALARMS_WARNINGS".SERVICES."708118" := #U02_LOWER_TABLE_PRESSURIZATION_ALARM;
END_REGION

REGION Network 54: UNIT 02 LOWER TABLE PRESSURIZATION SWITCH ALARM
   RUNG wire#powerrail
      Contact( #PRESSURE_OFF_DELAYED )
      Contact( #U02_UPPER_TABLE_PRESSURIZED )
      wire#w1
      Contact( #O_BYTE_1.U02_LOWER_TABLE_PRESSURIZED )
      wire#w2
      Coil( #U02_LOWER_TABLE_PRESSURIZATION_SWITCH_ALARM )
   END_RUNG
   RUNG wire#powerrail
      Contact( #U02_LOWER_TABLE_PRESSURIZATION_SWITCH_ALARM )
      I_Contact( "DB2120_MPP_ITC_IPC".RESET_FAULTS )
   END_RUNG wire#w1
   RUNG wire#w2
      Coil( "DB426_ALARMS_WARNINGS".SERVICES."708119" )
   END_RUNG
   // the same network as SCL:
   #U02_LOWER_TABLE_PRESSURIZATION_SWITCH_ALARM := ((#PRESSURE_OFF_DELAYED AND #U02_UPPER_TABLE_PRESSURIZED) OR (#U02_LOWER_TABLE_PRESSURIZATION_SWITCH_ALARM AND NOT "DB2120_MPP_ITC_IPC".RESET_FAULTS)) AND #O_BYTE_1.U02_LOWER_TABLE_PRESSURIZED;
   "DB426_ALARMS_WARNINGS".SERVICES."708119" := #U02_LOWER_TABLE_PRESSURIZATION_SWITCH_ALARM;
END_REGION

REGION Network 55: UNIT 02 CART AXIS X PRESSURIZATION ALARM
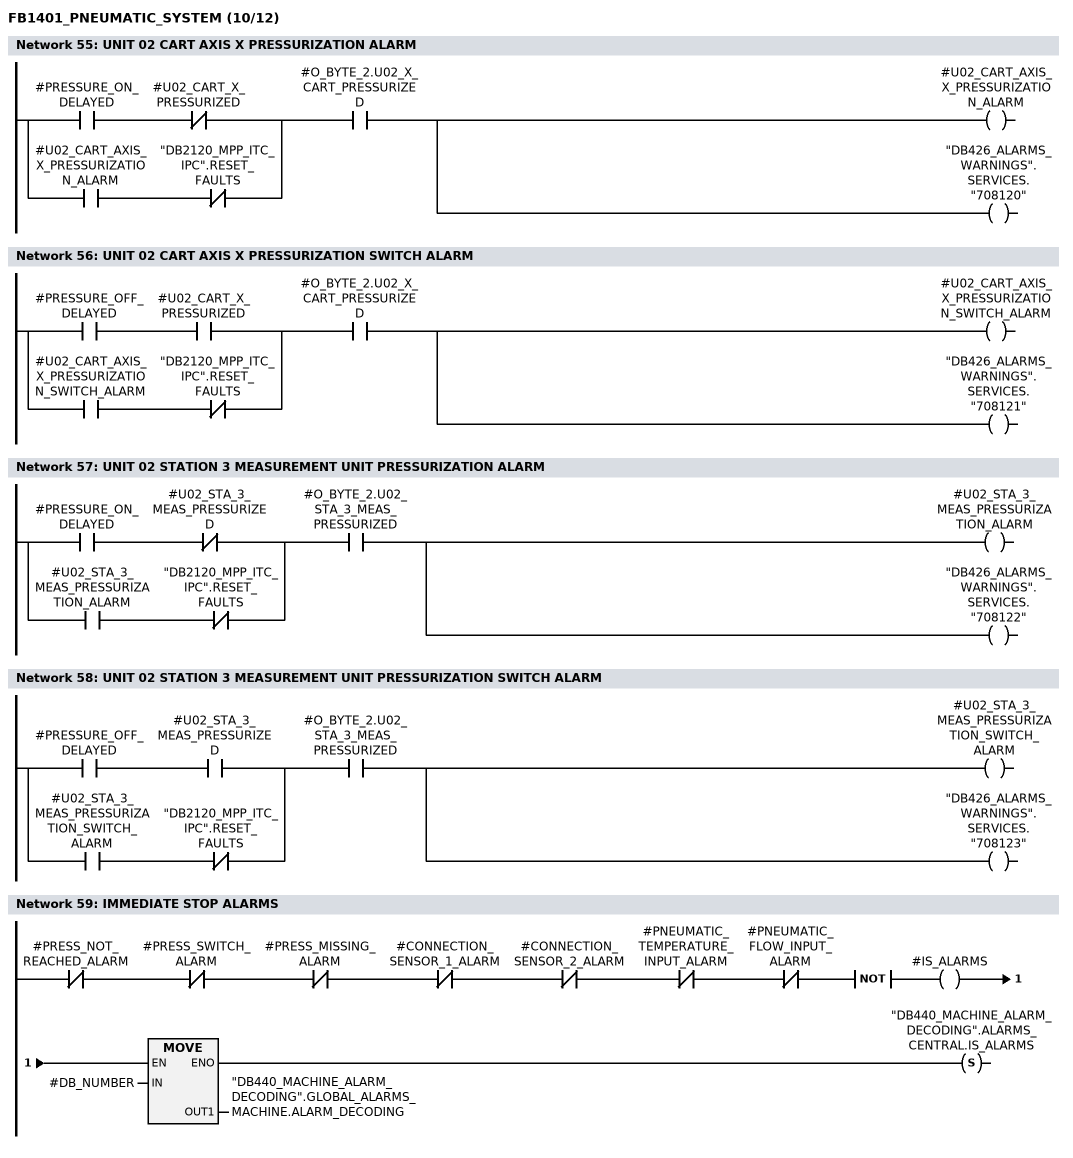
   RUNG wire#powerrail
      Contact( #PRESSURE_ON_DELAYED )
      I_Contact( #U02_CART_X_PRESSURIZED )
      wire#w1
      Contact( #O_BYTE_2.U02_X_CART_PRESSURIZED )
      wire#w2
      Coil( #U02_CART_AXIS_X_PRESSURIZATION_ALARM )
   END_RUNG
   RUNG wire#powerrail
      Contact( #U02_CART_AXIS_X_PRESSURIZATION_ALARM )
      I_Contact( "DB2120_MPP_ITC_IPC".RESET_FAULTS )
   END_RUNG wire#w1
   RUNG wire#w2
      Coil( "DB426_ALARMS_WARNINGS".SERVICES."708120" )
   END_RUNG
   // the same network as SCL:
   #U02_CART_AXIS_X_PRESSURIZATION_ALARM := ((#PRESSURE_ON_DELAYED AND NOT #U02_CART_X_PRESSURIZED) OR (#U02_CART_AXIS_X_PRESSURIZATION_ALARM AND NOT "DB2120_MPP_ITC_IPC".RESET_FAULTS)) AND #O_BYTE_2.U02_X_CART_PRESSURIZED;
   "DB426_ALARMS_WARNINGS".SERVICES."708120" := #U02_CART_AXIS_X_PRESSURIZATION_ALARM;
END_REGION

REGION Network 56: UNIT 02 CART AXIS X PRESSURIZATION SWITCH ALARM
   RUNG wire#powerrail
      Contact( #PRESSURE_OFF_DELAYED )
      Contact( #U02_CART_X_PRESSURIZED )
      wire#w1
      Contact( #O_BYTE_2.U02_X_CART_PRESSURIZED )
      wire#w2
      Coil( #U02_CART_AXIS_X_PRESSURIZATION_SWITCH_ALARM )
   END_RUNG
   RUNG wire#powerrail
      Contact( #U02_CART_AXIS_X_PRESSURIZATION_SWITCH_ALARM )
      I_Contact( "DB2120_MPP_ITC_IPC".RESET_FAULTS )
   END_RUNG wire#w1
   RUNG wire#w2
      Coil( "DB426_ALARMS_WARNINGS".SERVICES."708121" )
   END_RUNG
   // the same network as SCL:
   #U02_CART_AXIS_X_PRESSURIZATION_SWITCH_ALARM := ((#PRESSURE_OFF_DELAYED AND #U02_CART_X_PRESSURIZED) OR (#U02_CART_AXIS_X_PRESSURIZATION_SWITCH_ALARM AND NOT "DB2120_MPP_ITC_IPC".RESET_FAULTS)) AND #O_BYTE_2.U02_X_CART_PRESSURIZED;
   "DB426_ALARMS_WARNINGS".SERVICES."708121" := #U02_CART_AXIS_X_PRESSURIZATION_SWITCH_ALARM;
END_REGION

REGION Network 57: UNIT 02 STATION 3 MEASUREMENT UNIT PRESSURIZATION ALARM
   RUNG wire#powerrail
      Contact( #PRESSURE_ON_DELAYED )
      I_Contact( #U02_STA_3_MEAS_PRESSURIZED )
      wire#w1
      Contact( #O_BYTE_2.U02_STA_3_MEAS_PRESSURIZED )
      wire#w2
      Coil( #U02_STA_3_MEAS_PRESSURIZATION_ALARM )
   END_RUNG
   RUNG wire#powerrail
      Contact( #U02_STA_3_MEAS_PRESSURIZATION_ALARM )
      I_Contact( "DB2120_MPP_ITC_IPC".RESET_FAULTS )
   END_RUNG wire#w1
   RUNG wire#w2
      Coil( "DB426_ALARMS_WARNINGS".SERVICES."708122" )
   END_RUNG
   // the same network as SCL:
   #U02_STA_3_MEAS_PRESSURIZATION_ALARM := ((#PRESSURE_ON_DELAYED AND NOT #U02_STA_3_MEAS_PRESSURIZED) OR (#U02_STA_3_MEAS_PRESSURIZATION_ALARM AND NOT "DB2120_MPP_ITC_IPC".RESET_FAULTS)) AND #O_BYTE_2.U02_STA_3_MEAS_PRESSURIZED;
   "DB426_ALARMS_WARNINGS".SERVICES."708122" := #U02_STA_3_MEAS_PRESSURIZATION_ALARM;
END_REGION

REGION Network 58: UNIT 02 STATION 3 MEASUREMENT UNIT PRESSURIZATION SWITCH ALARM
   RUNG wire#powerrail
      Contact( #PRESSURE_OFF_DELAYED )
      Contact( #U02_STA_3_MEAS_PRESSURIZED )
      wire#w1
      Contact( #O_BYTE_2.U02_STA_3_MEAS_PRESSURIZED )
      wire#w2
      Coil( #U02_STA_3_MEAS_PRESSURIZATION_SWITCH_ALARM )
   END_RUNG
   RUNG wire#powerrail
      Contact( #U02_STA_3_MEAS_PRESSURIZATION_SWITCH_ALARM )
      I_Contact( "DB2120_MPP_ITC_IPC".RESET_FAULTS )
   END_RUNG wire#w1
   RUNG wire#w2
      Coil( "DB426_ALARMS_WARNINGS".SERVICES."708123" )
   END_RUNG
   // the same network as SCL:
   #U02_STA_3_MEAS_PRESSURIZATION_SWITCH_ALARM := ((#PRESSURE_OFF_DELAYED AND #U02_STA_3_MEAS_PRESSURIZED) OR (#U02_STA_3_MEAS_PRESSURIZATION_SWITCH_ALARM AND NOT "DB2120_MPP_ITC_IPC".RESET_FAULTS)) AND #O_BYTE_2.U02_STA_3_MEAS_PRESSURIZED;
   "DB426_ALARMS_WARNINGS".SERVICES."708123" := #U02_STA_3_MEAS_PRESSURIZATION_SWITCH_ALARM;
END_REGION

REGION Network 59: IMMEDIATE STOP ALARMS
   RUNG wire#powerrail
      I_Contact( #PRESS_NOT_REACHED_ALARM )
      I_Contact( #PRESS_SWITCH_ALARM )
      I_Contact( #PRESS_MISSING_ALARM )
      I_Contact( #CONNECTION_SENSOR_1_ALARM )
      I_Contact( #CONNECTION_SENSOR_2_ALARM )
      I_Contact( #PNEUMATIC_TEMPERATURE_INPUT_ALARM )
      I_Contact( #PNEUMATIC_FLOW_INPUT_ALARM )
      Not()
      Coil( #IS_ALARMS )
      Move(in := #DB_NUMBER, out1 => "DB440_MACHINE_ALARM_DECODING".GLOBAL_ALARMS_MACHINE.ALARM_DECODING)
      S_Coil( "DB440_MACHINE_ALARM_DECODING".ALARMS_CENTRAL.IS_ALARMS )
   END_RUNG
   // the same network as SCL:
   #IS_ALARMS := NOT (NOT #PRESS_NOT_REACHED_ALARM AND NOT #PRESS_SWITCH_ALARM AND NOT #PRESS_MISSING_ALARM AND NOT #CONNECTION_SENSOR_1_ALARM AND NOT #CONNECTION_SENSOR_2_ALARM AND NOT #PNEUMATIC_TEMPERATURE_INPUT_ALARM AND NOT #PNEUMATIC_FLOW_INPUT_ALARM);
   IF #IS_ALARMS THEN
       "DB440_MACHINE_ALARM_DECODING".GLOBAL_ALARMS_MACHINE.ALARM_DECODING := #DB_NUMBER;
       "DB440_MACHINE_ALARM_DECODING".ALARMS_CENTRAL.IS_ALARMS := TRUE;
   END_IF;
END_REGION

REGION Network 60: STOP END OF CYCLE ALARMS
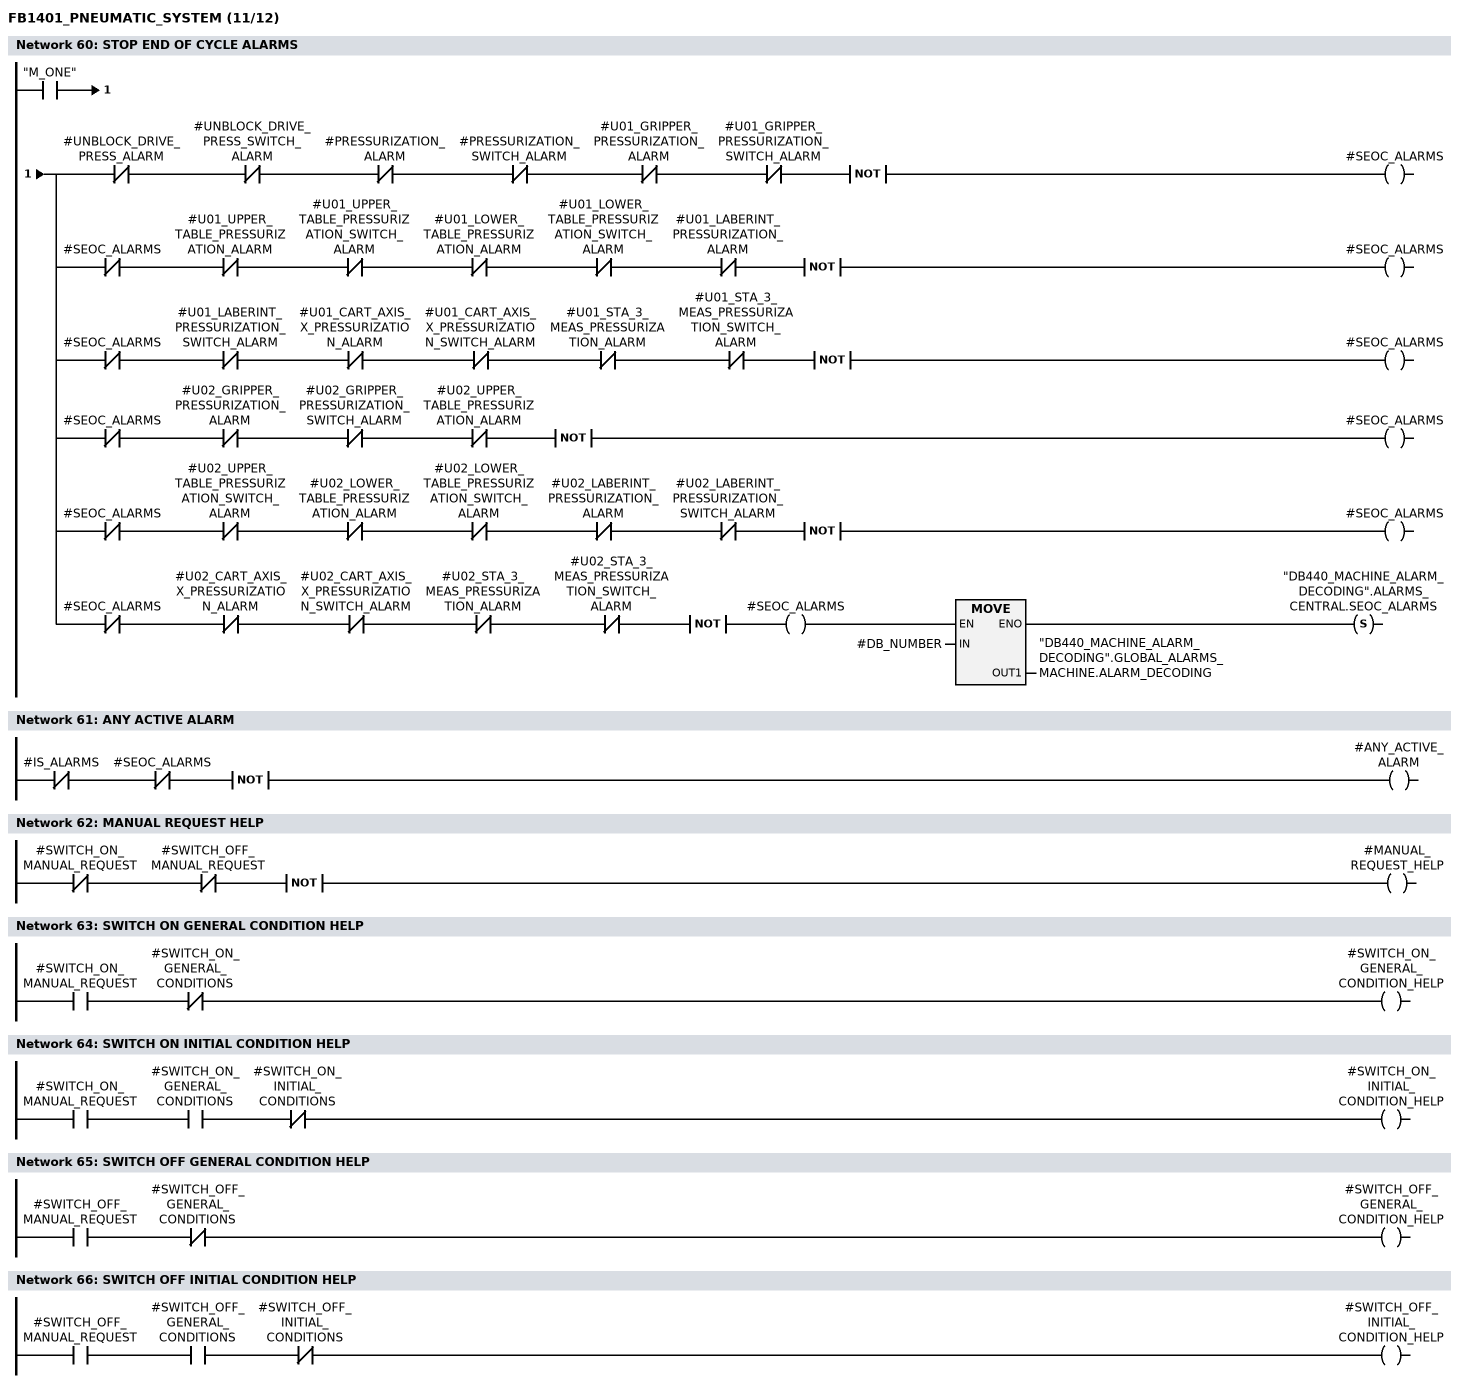
   RUNG wire#powerrail
      Contact( "M_ONE" )
      wire#w1
      I_Contact( #UNBLOCK_DRIVE_PRESS_ALARM )
      I_Contact( #UNBLOCK_DRIVE_PRESS_SWITCH_ALARM )
      I_Contact( #PRESSURIZATION_ALARM )
      I_Contact( #PRESSURIZATION_SWITCH_ALARM )
      I_Contact( #U01_GRIPPER_PRESSURIZATION_ALARM )
      I_Contact( #U01_GRIPPER_PRESSURIZATION_SWITCH_ALARM )
      Not()
      Coil( #SEOC_ALARMS )
   END_RUNG
   RUNG wire#w1
      I_Contact( #SEOC_ALARMS )
      I_Contact( #U01_UPPER_TABLE_PRESSURIZATION_ALARM )
      I_Contact( #U01_UPPER_TABLE_PRESSURIZATION_SWITCH_ALARM )
      I_Contact( #U01_LOWER_TABLE_PRESSURIZATION_ALARM )
      I_Contact( #U01_LOWER_TABLE_PRESSURIZATION_SWITCH_ALARM )
      I_Contact( #U01_LABERINT_PRESSURIZATION_ALARM )
      Not()
      Coil( #SEOC_ALARMS )
   END_RUNG
   RUNG wire#w1
      I_Contact( #SEOC_ALARMS )
      I_Contact( #U01_LABERINT_PRESSURIZATION_SWITCH_ALARM )
      I_Contact( #U01_CART_AXIS_X_PRESSURIZATION_ALARM )
      I_Contact( #U01_CART_AXIS_X_PRESSURIZATION_SWITCH_ALARM )
      I_Contact( #U01_STA_3_MEAS_PRESSURIZATION_ALARM )
      I_Contact( #U01_STA_3_MEAS_PRESSURIZATION_SWITCH_ALARM )
      Not()
      Coil( #SEOC_ALARMS )
   END_RUNG
   RUNG wire#w1
      I_Contact( #SEOC_ALARMS )
      I_Contact( #U02_GRIPPER_PRESSURIZATION_ALARM )
      I_Contact( #U02_GRIPPER_PRESSURIZATION_SWITCH_ALARM )
      I_Contact( #U02_UPPER_TABLE_PRESSURIZATION_ALARM )
      Not()
      Coil( #SEOC_ALARMS )
   END_RUNG
   RUNG wire#w1
      I_Contact( #SEOC_ALARMS )
      I_Contact( #U02_UPPER_TABLE_PRESSURIZATION_SWITCH_ALARM )
      I_Contact( #U02_LOWER_TABLE_PRESSURIZATION_ALARM )
      I_Contact( #U02_LOWER_TABLE_PRESSURIZATION_SWITCH_ALARM )
      I_Contact( #U02_LABERINT_PRESSURIZATION_ALARM )
      I_Contact( #U02_LABERINT_PRESSURIZATION_SWITCH_ALARM )
      Not()
      Coil( #SEOC_ALARMS )
   END_RUNG
   RUNG wire#w1
      I_Contact( #SEOC_ALARMS )
      I_Contact( #U02_CART_AXIS_X_PRESSURIZATION_ALARM )
      I_Contact( #U02_CART_AXIS_X_PRESSURIZATION_SWITCH_ALARM )
      I_Contact( #U02_STA_3_MEAS_PRESSURIZATION_ALARM )
      I_Contact( #U02_STA_3_MEAS_PRESSURIZATION_SWITCH_ALARM )
      Not()
      Coil( #SEOC_ALARMS )
      Move(in := #DB_NUMBER, out1 => "DB440_MACHINE_ALARM_DECODING".GLOBAL_ALARMS_MACHINE.ALARM_DECODING)
      S_Coil( "DB440_MACHINE_ALARM_DECODING".ALARMS_CENTRAL.SEOC_ALARMS )
   END_RUNG
   // the same network as SCL:
   #SEOC_ALARMS := NOT ("M_ONE" AND NOT #UNBLOCK_DRIVE_PRESS_ALARM AND NOT #UNBLOCK_DRIVE_PRESS_SWITCH_ALARM AND NOT #PRESSURIZATION_ALARM AND NOT #PRESSURIZATION_SWITCH_ALARM AND NOT #U01_GRIPPER_PRESSURIZATION_ALARM AND NOT #U01_GRIPPER_PRESSURIZATION_SWITCH_ALARM);
   #SEOC_ALARMS := NOT ("M_ONE" AND NOT #SEOC_ALARMS AND NOT #U01_UPPER_TABLE_PRESSURIZATION_ALARM AND NOT #U01_UPPER_TABLE_PRESSURIZATION_SWITCH_ALARM AND NOT #U01_LOWER_TABLE_PRESSURIZATION_ALARM AND NOT #U01_LOWER_TABLE_PRESSURIZATION_SWITCH_ALARM AND NOT #U01_LABERINT_PRESSURIZATION_ALARM);
   #SEOC_ALARMS := NOT ("M_ONE" AND NOT #SEOC_ALARMS AND NOT #U01_LABERINT_PRESSURIZATION_SWITCH_ALARM AND NOT #U01_CART_AXIS_X_PRESSURIZATION_ALARM AND NOT #U01_CART_AXIS_X_PRESSURIZATION_SWITCH_ALARM AND NOT #U01_STA_3_MEAS_PRESSURIZATION_ALARM AND NOT #U01_STA_3_MEAS_PRESSURIZATION_SWITCH_ALARM);
   #SEOC_ALARMS := NOT ("M_ONE" AND NOT #SEOC_ALARMS AND NOT #U02_GRIPPER_PRESSURIZATION_ALARM AND NOT #U02_GRIPPER_PRESSURIZATION_SWITCH_ALARM AND NOT #U02_UPPER_TABLE_PRESSURIZATION_ALARM);
   #SEOC_ALARMS := NOT ("M_ONE" AND NOT #SEOC_ALARMS AND NOT #U02_UPPER_TABLE_PRESSURIZATION_SWITCH_ALARM AND NOT #U02_LOWER_TABLE_PRESSURIZATION_ALARM AND NOT #U02_LOWER_TABLE_PRESSURIZATION_SWITCH_ALARM AND NOT #U02_LABERINT_PRESSURIZATION_ALARM AND NOT #U02_LABERINT_PRESSURIZATION_SWITCH_ALARM);
   #SEOC_ALARMS := NOT ("M_ONE" AND NOT #SEOC_ALARMS AND NOT #U02_CART_AXIS_X_PRESSURIZATION_ALARM AND NOT #U02_CART_AXIS_X_PRESSURIZATION_SWITCH_ALARM AND NOT #U02_STA_3_MEAS_PRESSURIZATION_ALARM AND NOT #U02_STA_3_MEAS_PRESSURIZATION_SWITCH_ALARM);
   IF #SEOC_ALARMS THEN
       "DB440_MACHINE_ALARM_DECODING".GLOBAL_ALARMS_MACHINE.ALARM_DECODING := #DB_NUMBER;
       "DB440_MACHINE_ALARM_DECODING".ALARMS_CENTRAL.SEOC_ALARMS := TRUE;
   END_IF;
END_REGION

REGION Network 61: ANY ACTIVE ALARM
   RUNG wire#powerrail
      I_Contact( #IS_ALARMS )
      I_Contact( #SEOC_ALARMS )
      Not()
      Coil( #ANY_ACTIVE_ALARM )
   END_RUNG
   // the same network as SCL:
   #ANY_ACTIVE_ALARM := NOT (NOT #IS_ALARMS AND NOT #SEOC_ALARMS);
END_REGION

REGION Network 62: MANUAL REQUEST HELP
   RUNG wire#powerrail
      I_Contact( #SWITCH_ON_MANUAL_REQUEST )
      I_Contact( #SWITCH_OFF_MANUAL_REQUEST )
      Not()
      Coil( #MANUAL_REQUEST_HELP )
   END_RUNG
   // the same network as SCL:
   #MANUAL_REQUEST_HELP := NOT (NOT #SWITCH_ON_MANUAL_REQUEST AND NOT #SWITCH_OFF_MANUAL_REQUEST);
END_REGION

REGION Network 63: SWITCH ON GENERAL CONDITION HELP
   RUNG wire#powerrail
      Contact( #SWITCH_ON_MANUAL_REQUEST )
      I_Contact( #SWITCH_ON_GENERAL_CONDITIONS )
      Coil( #SWITCH_ON_GENERAL_CONDITION_HELP )
   END_RUNG
   // the same network as SCL:
   #SWITCH_ON_GENERAL_CONDITION_HELP := #SWITCH_ON_MANUAL_REQUEST AND NOT #SWITCH_ON_GENERAL_CONDITIONS;
END_REGION

REGION Network 64: SWITCH ON INITIAL CONDITION HELP
   RUNG wire#powerrail
      Contact( #SWITCH_ON_MANUAL_REQUEST )
      Contact( #SWITCH_ON_GENERAL_CONDITIONS )
      I_Contact( #SWITCH_ON_INITIAL_CONDITIONS )
      Coil( #SWITCH_ON_INITIAL_CONDITION_HELP )
   END_RUNG
   // the same network as SCL:
   #SWITCH_ON_INITIAL_CONDITION_HELP := #SWITCH_ON_MANUAL_REQUEST AND #SWITCH_ON_GENERAL_CONDITIONS AND NOT #SWITCH_ON_INITIAL_CONDITIONS;
END_REGION

REGION Network 65: SWITCH OFF GENERAL CONDITION HELP
   RUNG wire#powerrail
      Contact( #SWITCH_OFF_MANUAL_REQUEST )
      I_Contact( #SWITCH_OFF_GENERAL_CONDITIONS )
      Coil( #SWITCH_OFF_GENERAL_CONDITION_HELP )
   END_RUNG
   // the same network as SCL:
   #SWITCH_OFF_GENERAL_CONDITION_HELP := #SWITCH_OFF_MANUAL_REQUEST AND NOT #SWITCH_OFF_GENERAL_CONDITIONS;
END_REGION

REGION Network 66: SWITCH OFF INITIAL CONDITION HELP
   RUNG wire#powerrail
      Contact( #SWITCH_OFF_MANUAL_REQUEST )
      Contact( #SWITCH_OFF_GENERAL_CONDITIONS )
      I_Contact( #SWITCH_OFF_INITIAL_CONDITIONS )
      Coil( #SWITCH_OFF_INITIAL_CONDITION_HELP )
   END_RUNG
   // the same network as SCL:
   #SWITCH_OFF_INITIAL_CONDITION_HELP := #SWITCH_OFF_MANUAL_REQUEST AND #SWITCH_OFF_GENERAL_CONDITIONS AND NOT #SWITCH_OFF_INITIAL_CONDITIONS;
END_REGION

REGION Network 67: HMI STATUS / HMI REACHED POSITION
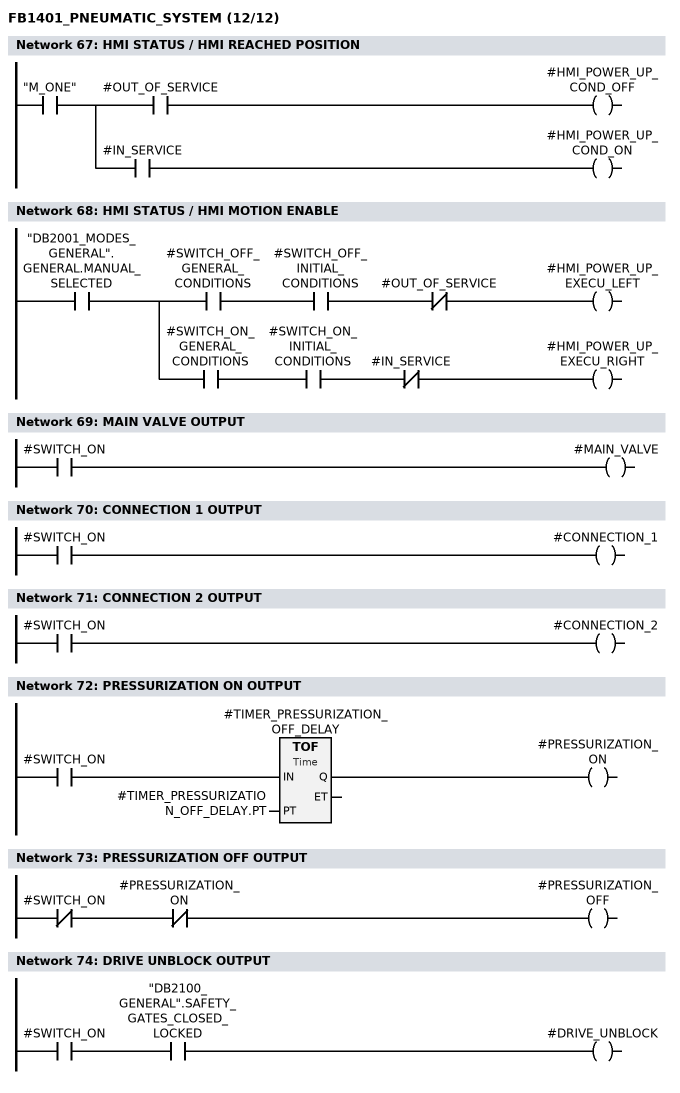
   RUNG wire#powerrail
      Contact( "M_ONE" )
      wire#w1
      Contact( #OUT_OF_SERVICE )
      Coil( #HMI_POWER_UP_COND_OFF )
   END_RUNG
   RUNG wire#w1
      Contact( #IN_SERVICE )
      Coil( #HMI_POWER_UP_COND_ON )
   END_RUNG
   // the same network as SCL:
   #HMI_POWER_UP_COND_OFF := "M_ONE" AND #OUT_OF_SERVICE;
   #HMI_POWER_UP_COND_ON := "M_ONE" AND #IN_SERVICE;
END_REGION

REGION Network 68: HMI STATUS / HMI MOTION ENABLE
   RUNG wire#powerrail
      Contact( "DB2001_MODES_GENERAL".GENERAL.MANUAL_SELECTED )
      wire#w1
      Contact( #SWITCH_OFF_GENERAL_CONDITIONS )
      Contact( #SWITCH_OFF_INITIAL_CONDITIONS )
      I_Contact( #OUT_OF_SERVICE )
      Coil( #HMI_POWER_UP_EXECU_LEFT )
   END_RUNG
   RUNG wire#w1
      Contact( #SWITCH_ON_GENERAL_CONDITIONS )
      Contact( #SWITCH_ON_INITIAL_CONDITIONS )
      I_Contact( #IN_SERVICE )
      Coil( #HMI_POWER_UP_EXECU_RIGHT )
   END_RUNG
   // the same network as SCL:
   #HMI_POWER_UP_EXECU_LEFT := "DB2001_MODES_GENERAL".GENERAL.MANUAL_SELECTED AND #SWITCH_OFF_GENERAL_CONDITIONS AND #SWITCH_OFF_INITIAL_CONDITIONS AND NOT #OUT_OF_SERVICE;
   #HMI_POWER_UP_EXECU_RIGHT := "DB2001_MODES_GENERAL".GENERAL.MANUAL_SELECTED AND #SWITCH_ON_GENERAL_CONDITIONS AND #SWITCH_ON_INITIAL_CONDITIONS AND NOT #IN_SERVICE;
END_REGION

REGION Network 69: MAIN VALVE OUTPUT
   RUNG wire#powerrail
      Contact( #SWITCH_ON )
      Coil( #MAIN_VALVE )
   END_RUNG
   // the same network as SCL:
   #MAIN_VALVE := #SWITCH_ON;
END_REGION

REGION Network 70: CONNECTION 1 OUTPUT
   RUNG wire#powerrail
      Contact( #SWITCH_ON )
      Coil( #CONNECTION_1 )
   END_RUNG
   // the same network as SCL:
   #CONNECTION_1 := #SWITCH_ON;
END_REGION

REGION Network 71: CONNECTION 2 OUTPUT
   RUNG wire#powerrail
      Contact( #SWITCH_ON )
      Coil( #CONNECTION_2 )
   END_RUNG
   // the same network as SCL:
   #CONNECTION_2 := #SWITCH_ON;
END_REGION

REGION Network 72: PRESSURIZATION ON OUTPUT
   RUNG wire#powerrail
      Contact( #SWITCH_ON )
      { S7_Templates := "time_type := Time" } #TIMER_PRESSURIZATION_OFF_DELAY.TOF(pt := #TIMER_PRESSURIZATION_OFF_DELAY.PT, et =>)
      Coil( #PRESSURIZATION_ON )
   END_RUNG
   // the same network as SCL:
   #TIMER_PRESSURIZATION_OFF_DELAY(IN := #SWITCH_ON, PT := #TIMER_PRESSURIZATION_OFF_DELAY.PT);   // TOF
   #PRESSURIZATION_ON := #TIMER_PRESSURIZATION_OFF_DELAY.Q;
END_REGION

REGION Network 73: PRESSURIZATION OFF OUTPUT
   RUNG wire#powerrail
      I_Contact( #SWITCH_ON )
      I_Contact( #PRESSURIZATION_ON )
      Coil( #PRESSURIZATION_OFF )
   END_RUNG
   // the same network as SCL:
   #PRESSURIZATION_OFF := NOT #SWITCH_ON AND NOT #PRESSURIZATION_ON;
END_REGION

REGION Network 74: DRIVE UNBLOCK OUTPUT
   RUNG wire#powerrail
      Contact( #SWITCH_ON )
      Contact( "DB2100_GENERAL".SAFETY_GATES_CLOSED_LOCKED )
      Coil( #DRIVE_UNBLOCK )
   END_RUNG
   // the same network as SCL:
   #DRIVE_UNBLOCK := #SWITCH_ON AND "DB2100_GENERAL".SAFETY_GATES_CLOSED_LOCKED;
END_REGION
END_FUNCTION_BLOCK
